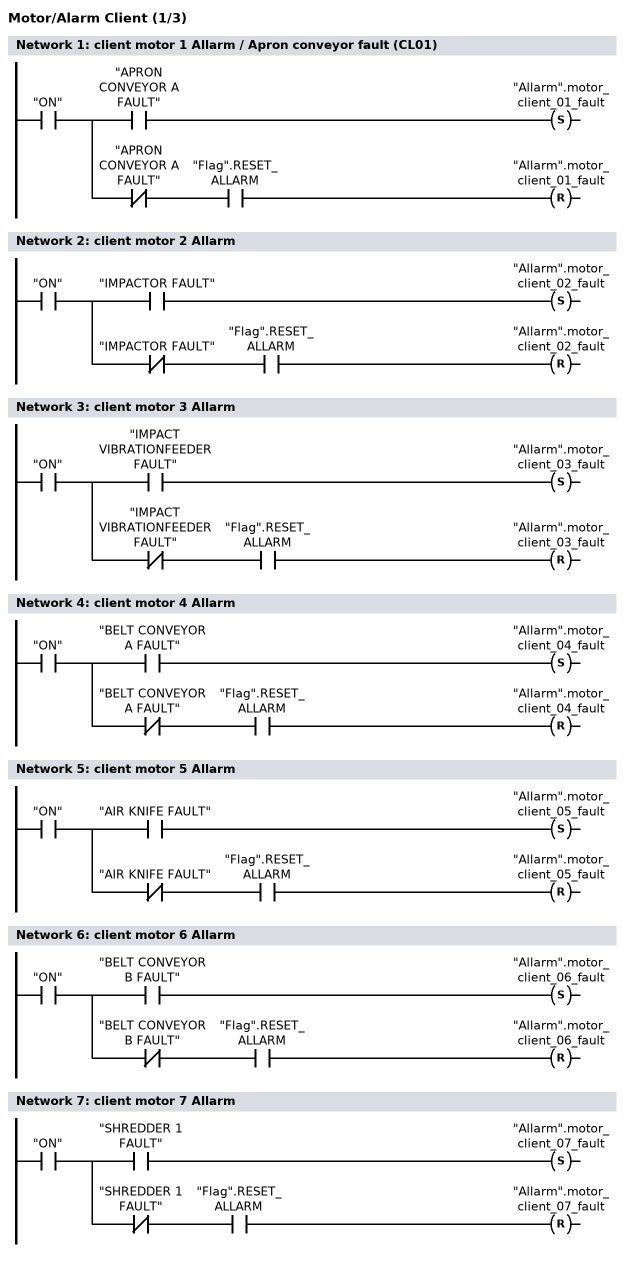
   RUNG wire#powerrail
      Contact( "ON" )
      wire#w1
      Contact( "APRON CONVEYOR A FAULT" )
      S_Coil( "Allarm".motor_client_01_fault )
   END_RUNG
   RUNG wire#w1
      I_Contact( "APRON CONVEYOR A FAULT" )
      Contact( "Flag".RESET_ALLARM )
      R_Coil( "Allarm".motor_client_01_fault )
   END_RUNG
   // the same network as SCL:
   IF "ON" AND "APRON CONVEYOR A FAULT" THEN "Allarm".motor_client_01_fault := TRUE; END_IF;
   IF "ON" AND NOT "APRON CONVEYOR A FAULT" AND "Flag".RESET_ALLARM THEN
       "Allarm".motor_client_01_fault := FALSE;
   END_IF;
END_REGION

REGION Network 2: client motor 2 Allarm
   RUNG wire#powerrail
      Contact( "ON" )
      wire#w1
      Contact( "IMPACTOR FAULT" )
      S_Coil( "Allarm".motor_client_02_fault )
   END_RUNG
   RUNG wire#w1
      I_Contact( "IMPACTOR FAULT" )
      Contact( "Flag".RESET_ALLARM )
      R_Coil( "Allarm".motor_client_02_fault )
   END_RUNG
   // the same network as SCL:
   IF "ON" AND "IMPACTOR FAULT" THEN "Allarm".motor_client_02_fault := TRUE; END_IF;
   IF "ON" AND NOT "IMPACTOR FAULT" AND "Flag".RESET_ALLARM THEN
       "Allarm".motor_client_02_fault := FALSE;
   END_IF;
END_REGION

REGION Network 3: client motor 3 Allarm
   RUNG wire#powerrail
      Contact( "ON" )
      wire#w1
      Contact( "IMPACT VIBRATIONFEEDER FAULT" )
      S_Coil( "Allarm".motor_client_03_fault )
   END_RUNG
   RUNG wire#w1
      I_Contact( "IMPACT VIBRATIONFEEDER FAULT" )
      Contact( "Flag".RESET_ALLARM )
      R_Coil( "Allarm".motor_client_03_fault )
   END_RUNG
   // the same network as SCL:
   IF "ON" AND "IMPACT VIBRATIONFEEDER FAULT" THEN "Allarm".motor_client_03_fault := TRUE; END_IF;
   IF "ON" AND NOT "IMPACT VIBRATIONFEEDER FAULT" AND "Flag".RESET_ALLARM THEN
       "Allarm".motor_client_03_fault := FALSE;
   END_IF;
END_REGION

REGION Network 4: client motor 4 Allarm
   RUNG wire#powerrail
      Contact( "ON" )
      wire#w1
      Contact( "BELT CONVEYOR  A FAULT" )
      S_Coil( "Allarm".motor_client_04_fault )
   END_RUNG
   RUNG wire#w1
      I_Contact( "BELT CONVEYOR  A FAULT" )
      Contact( "Flag".RESET_ALLARM )
      R_Coil( "Allarm".motor_client_04_fault )
   END_RUNG
   // the same network as SCL:
   IF "ON" AND "BELT CONVEYOR  A FAULT" THEN "Allarm".motor_client_04_fault := TRUE; END_IF;
   IF "ON" AND NOT "BELT CONVEYOR  A FAULT" AND "Flag".RESET_ALLARM THEN
       "Allarm".motor_client_04_fault := FALSE;
   END_IF;
END_REGION

REGION Network 5: client motor 5 Allarm
   RUNG wire#powerrail
      Contact( "ON" )
      wire#w1
      Contact( "AIR KNIFE FAULT" )
      S_Coil( "Allarm".motor_client_05_fault )
   END_RUNG
   RUNG wire#w1
      I_Contact( "AIR KNIFE FAULT" )
      Contact( "Flag".RESET_ALLARM )
      R_Coil( "Allarm".motor_client_05_fault )
   END_RUNG
   // the same network as SCL:
   IF "ON" AND "AIR KNIFE FAULT" THEN "Allarm".motor_client_05_fault := TRUE; END_IF;
   IF "ON" AND NOT "AIR KNIFE FAULT" AND "Flag".RESET_ALLARM THEN
       "Allarm".motor_client_05_fault := FALSE;
   END_IF;
END_REGION

REGION Network 6: client motor 6 Allarm
   RUNG wire#powerrail
      Contact( "ON" )
      wire#w1
      Contact( "BELT CONVEYOR B FAULT" )
      S_Coil( "Allarm".motor_client_06_fault )
   END_RUNG
   RUNG wire#w1
      I_Contact( "BELT CONVEYOR B FAULT" )
      Contact( "Flag".RESET_ALLARM )
      R_Coil( "Allarm".motor_client_06_fault )
   END_RUNG
   // the same network as SCL:
   IF "ON" AND "BELT CONVEYOR B FAULT" THEN "Allarm".motor_client_06_fault := TRUE; END_IF;
   IF "ON" AND NOT "BELT CONVEYOR B FAULT" AND "Flag".RESET_ALLARM THEN
       "Allarm".motor_client_06_fault := FALSE;
   END_IF;
END_REGION

REGION Network 7: client motor 7 Allarm
   RUNG wire#powerrail
      Contact( "ON" )
      wire#w1
      Contact( "SHREDDER 1 FAULT" )
      S_Coil( "Allarm".motor_client_07_fault )
   END_RUNG
   RUNG wire#w1
      I_Contact( "SHREDDER 1 FAULT" )
      Contact( "Flag".RESET_ALLARM )
      R_Coil( "Allarm".motor_client_07_fault )
   END_RUNG
   // the same network as SCL:
   IF "ON" AND "SHREDDER 1 FAULT" THEN "Allarm".motor_client_07_fault := TRUE; END_IF;
   IF "ON" AND NOT "SHREDDER 1 FAULT" AND "Flag".RESET_ALLARM THEN
       "Allarm".motor_client_07_fault := FALSE;
   END_IF;
END_REGION

REGION Network 8: client motor 8 Allarm
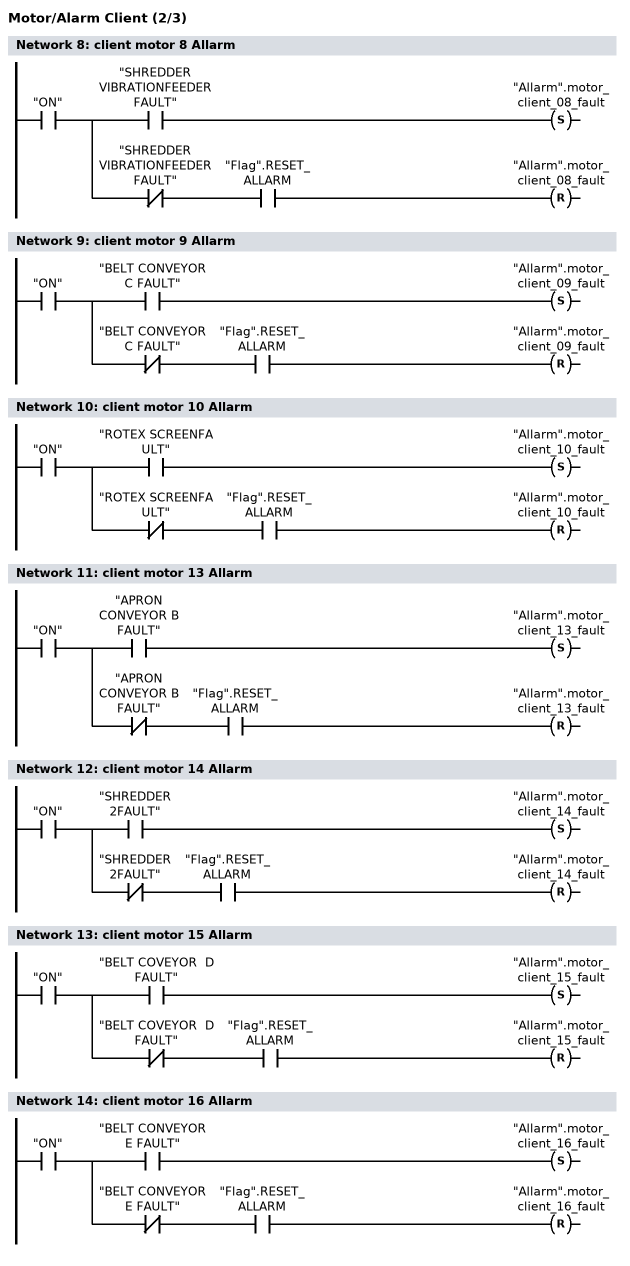
   RUNG wire#powerrail
      Contact( "ON" )
      wire#w1
      Contact( "SHREDDER VIBRATIONFEEDER FAULT" )
      S_Coil( "Allarm".motor_client_08_fault )
   END_RUNG
   RUNG wire#w1
      I_Contact( "SHREDDER VIBRATIONFEEDER FAULT" )
      Contact( "Flag".RESET_ALLARM )
      R_Coil( "Allarm".motor_client_08_fault )
   END_RUNG
   // the same network as SCL:
   IF "ON" AND "SHREDDER VIBRATIONFEEDER FAULT" THEN "Allarm".motor_client_08_fault := TRUE; END_IF;
   IF "ON" AND NOT "SHREDDER VIBRATIONFEEDER FAULT" AND "Flag".RESET_ALLARM THEN
       "Allarm".motor_client_08_fault := FALSE;
   END_IF;
END_REGION

REGION Network 9: client motor 9 Allarm
   RUNG wire#powerrail
      Contact( "ON" )
      wire#w1
      Contact( "BELT CONVEYOR C FAULT" )
      S_Coil( "Allarm".motor_client_09_fault )
   END_RUNG
   RUNG wire#w1
      I_Contact( "BELT CONVEYOR C FAULT" )
      Contact( "Flag".RESET_ALLARM )
      R_Coil( "Allarm".motor_client_09_fault )
   END_RUNG
   // the same network as SCL:
   IF "ON" AND "BELT CONVEYOR C FAULT" THEN "Allarm".motor_client_09_fault := TRUE; END_IF;
   IF "ON" AND NOT "BELT CONVEYOR C FAULT" AND "Flag".RESET_ALLARM THEN
       "Allarm".motor_client_09_fault := FALSE;
   END_IF;
END_REGION

REGION Network 10: client motor 10 Allarm
   RUNG wire#powerrail
      Contact( "ON" )
      wire#w1
      Contact( "ROTEX SCREENFAULT" )
      S_Coil( "Allarm".motor_client_10_fault )
   END_RUNG
   RUNG wire#w1
      I_Contact( "ROTEX SCREENFAULT" )
      Contact( "Flag".RESET_ALLARM )
      R_Coil( "Allarm".motor_client_10_fault )
   END_RUNG
   // the same network as SCL:
   IF "ON" AND "ROTEX SCREENFAULT" THEN "Allarm".motor_client_10_fault := TRUE; END_IF;
   IF "ON" AND NOT "ROTEX SCREENFAULT" AND "Flag".RESET_ALLARM THEN
       "Allarm".motor_client_10_fault := FALSE;
   END_IF;
END_REGION

REGION Network 11: client motor 13 Allarm
   RUNG wire#powerrail
      Contact( "ON" )
      wire#w1
      Contact( "APRON CONVEYOR B FAULT" )
      S_Coil( "Allarm".motor_client_13_fault )
   END_RUNG
   RUNG wire#w1
      I_Contact( "APRON CONVEYOR B FAULT" )
      Contact( "Flag".RESET_ALLARM )
      R_Coil( "Allarm".motor_client_13_fault )
   END_RUNG
   // the same network as SCL:
   IF "ON" AND "APRON CONVEYOR B FAULT" THEN "Allarm".motor_client_13_fault := TRUE; END_IF;
   IF "ON" AND NOT "APRON CONVEYOR B FAULT" AND "Flag".RESET_ALLARM THEN
       "Allarm".motor_client_13_fault := FALSE;
   END_IF;
END_REGION

REGION Network 12: client motor 14 Allarm
   RUNG wire#powerrail
      Contact( "ON" )
      wire#w1
      Contact( "SHREDDER 2FAULT" )
      S_Coil( "Allarm".motor_client_14_fault )
   END_RUNG
   RUNG wire#w1
      I_Contact( "SHREDDER 2FAULT" )
      Contact( "Flag".RESET_ALLARM )
      R_Coil( "Allarm".motor_client_14_fault )
   END_RUNG
   // the same network as SCL:
   IF "ON" AND "SHREDDER 2FAULT" THEN "Allarm".motor_client_14_fault := TRUE; END_IF;
   IF "ON" AND NOT "SHREDDER 2FAULT" AND "Flag".RESET_ALLARM THEN
       "Allarm".motor_client_14_fault := FALSE;
   END_IF;
END_REGION

REGION Network 13: client motor 15 Allarm
   RUNG wire#powerrail
      Contact( "ON" )
      wire#w1
      Contact( "BELT COVEYOR  D FAULT" )
      S_Coil( "Allarm".motor_client_15_fault )
   END_RUNG
   RUNG wire#w1
      I_Contact( "BELT COVEYOR  D FAULT" )
      Contact( "Flag".RESET_ALLARM )
      R_Coil( "Allarm".motor_client_15_fault )
   END_RUNG
   // the same network as SCL:
   IF "ON" AND "BELT COVEYOR  D FAULT" THEN "Allarm".motor_client_15_fault := TRUE; END_IF;
   IF "ON" AND NOT "BELT COVEYOR  D FAULT" AND "Flag".RESET_ALLARM THEN
       "Allarm".motor_client_15_fault := FALSE;
   END_IF;
END_REGION

REGION Network 14: client motor 16 Allarm
   RUNG wire#powerrail
      Contact( "ON" )
      wire#w1
      Contact( "BELT CONVEYOR  E FAULT" )
      S_Coil( "Allarm".motor_client_16_fault )
   END_RUNG
   RUNG wire#w1
      I_Contact( "BELT CONVEYOR  E FAULT" )
      Contact( "Flag".RESET_ALLARM )
      R_Coil( "Allarm".motor_client_16_fault )
   END_RUNG
   // the same network as SCL:
   IF "ON" AND "BELT CONVEYOR  E FAULT" THEN "Allarm".motor_client_16_fault := TRUE; END_IF;
   IF "ON" AND NOT "BELT CONVEYOR  E FAULT" AND "Flag".RESET_ALLARM THEN
       "Allarm".motor_client_16_fault := FALSE;
   END_IF;
END_REGION

REGION Network 15: client motor 17 Allarm
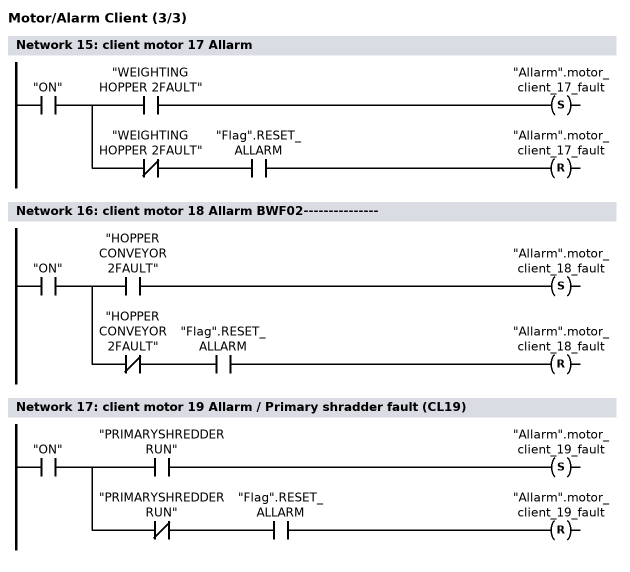
   RUNG wire#powerrail
      Contact( "ON" )
      wire#w1
      Contact( "WEIGHTING HOPPER 2FAULT" )
      S_Coil( "Allarm".motor_client_17_fault )
   END_RUNG
   RUNG wire#w1
      I_Contact( "WEIGHTING HOPPER 2FAULT" )
      Contact( "Flag".RESET_ALLARM )
      R_Coil( "Allarm".motor_client_17_fault )
   END_RUNG
   // the same network as SCL:
   IF "ON" AND "WEIGHTING HOPPER 2FAULT" THEN "Allarm".motor_client_17_fault := TRUE; END_IF;
   IF "ON" AND NOT "WEIGHTING HOPPER 2FAULT" AND "Flag".RESET_ALLARM THEN
       "Allarm".motor_client_17_fault := FALSE;
   END_IF;
END_REGION

REGION Network 16: client motor 18 Allarm BWF02---------------
   RUNG wire#powerrail
      Contact( "ON" )
      wire#w1
      Contact( "HOPPER CONVEYOR 2FAULT" )
      S_Coil( "Allarm".motor_client_18_fault )
   END_RUNG
   RUNG wire#w1
      I_Contact( "HOPPER CONVEYOR 2FAULT" )
      Contact( "Flag".RESET_ALLARM )
      R_Coil( "Allarm".motor_client_18_fault )
   END_RUNG
   // the same network as SCL:
   IF "ON" AND "HOPPER CONVEYOR 2FAULT" THEN "Allarm".motor_client_18_fault := TRUE; END_IF;
   IF "ON" AND NOT "HOPPER CONVEYOR 2FAULT" AND "Flag".RESET_ALLARM THEN
       "Allarm".motor_client_18_fault := FALSE;
   END_IF;
END_REGION

REGION Network 17: client motor 19 Allarm / Primary shradder fault (CL19)
   RUNG wire#powerrail
      Contact( "ON" )
      wire#w1
      Contact( "PRIMARYSHREDDER RUN" )
      S_Coil( "Allarm".motor_client_19_fault )
   END_RUNG
   RUNG wire#w1
      I_Contact( "PRIMARYSHREDDER RUN" )
      Contact( "Flag".RESET_ALLARM )
      R_Coil( "Allarm".motor_client_19_fault )
   END_RUNG
   // the same network as SCL:
   IF "ON" AND "PRIMARYSHREDDER RUN" THEN "Allarm".motor_client_19_fault := TRUE; END_IF;
   IF "ON" AND NOT "PRIMARYSHREDDER RUN" AND "Flag".RESET_ALLARM THEN
       "Allarm".motor_client_19_fault := FALSE;
   END_IF;
END_REGION
END_FUNCTION

FUNCTION "Burner Control" : Void   // FC12, LAD
TITLE = Burner allarms and control
{ S7_Optimized_Access := 'FALSE' }
VERSION : 0.1
   VAR_TEMP
      App00 : Int;
      App01 : Int;
      App02 : Int;
      App03 : Int;
   END_VAR
   VAR_TEMP   // added for the SCL form of the ladder/FBD networks
      _w1 : Bool;
      _w2 : Bool;
      _w3 : Bool;
      _w4 : Bool;
      _w5 : Bool;
      _w6 : Bool;
      _w7 : Bool;
      _w8 : Bool;
      _w9 : Bool;
      _w10 : Bool;
      _w11 : Bool;
   END_VAR
BEGIN

REGION Network 1: Burner box allarm / Burner control box FAULT
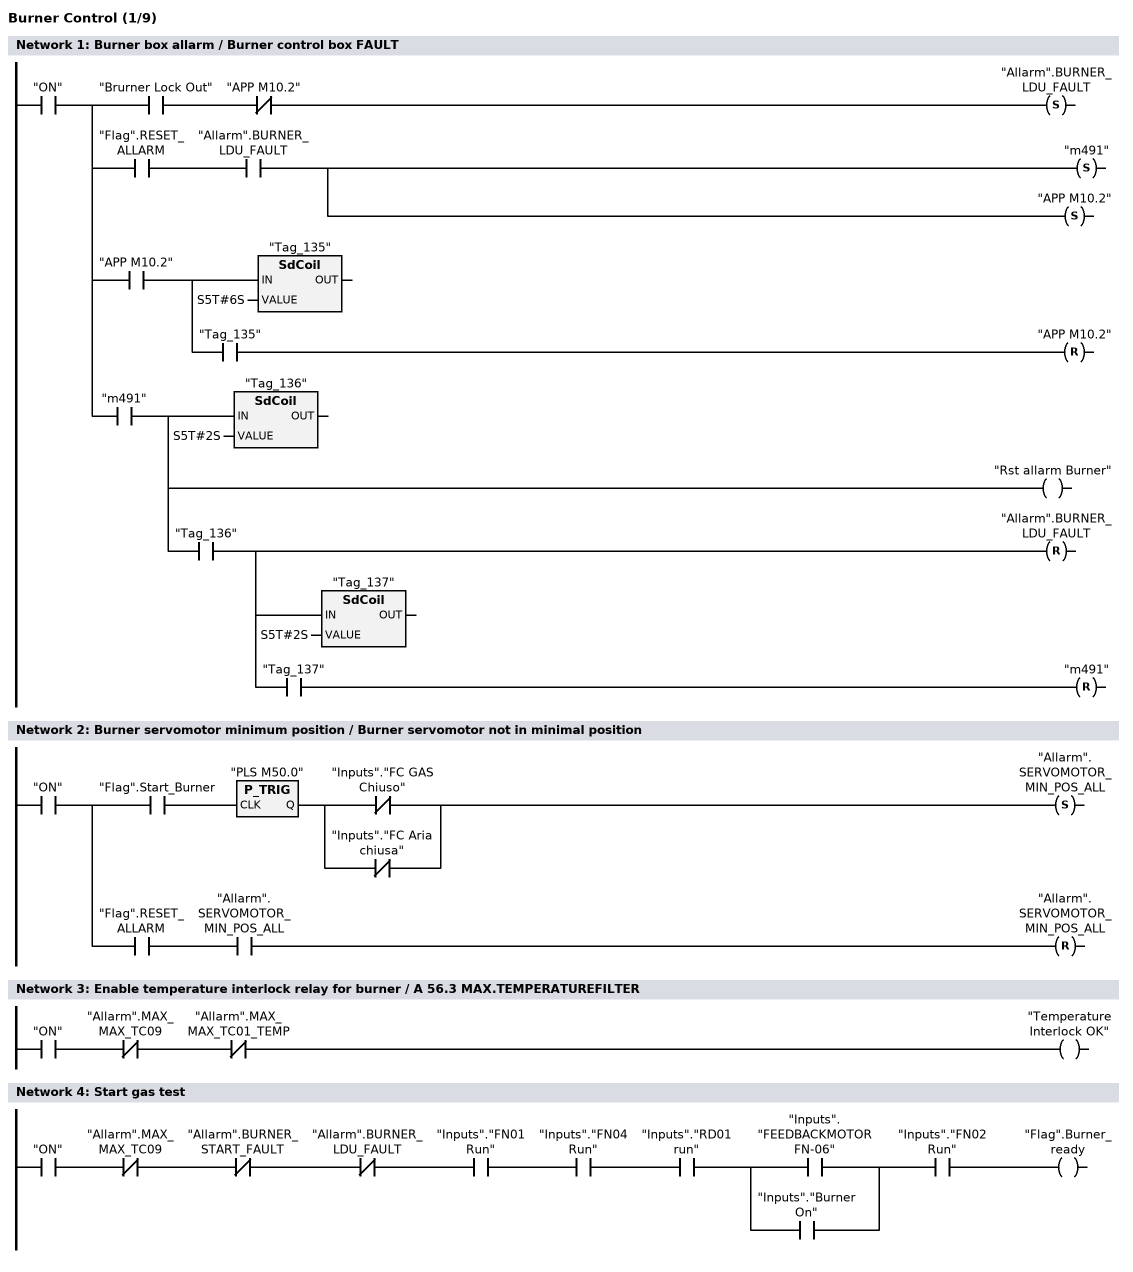
   // no SCL statement known for SdCoil: written as a call
   IF "ON" AND "Brurner Lock Out" AND NOT "APP M10.2" THEN "Allarm".BURNER_LDU_FAULT := TRUE; END_IF;
   IF "ON" AND "Flag".RESET_ALLARM AND "Allarm".BURNER_LDU_FAULT THEN
       "m491" := TRUE;
       "APP M10.2" := TRUE;
   END_IF;
   #_w1 := "ON" AND "APP M10.2";
   #_w2 := "ON";
   SdCoil(in := #_w1, value := S5T#6S, operand := "Tag_135");
   IF #_w1 AND "Tag_135" THEN "APP M10.2" := FALSE; END_IF;
   #_w3 := #_w2 AND "m491";
   SdCoil(in := #_w3, value := S5T#2S, operand := "Tag_136");
   "Rst allarm Burner" := #_w3;
   #_w4 := #_w3 AND "Tag_136";
   IF #_w4 THEN "Allarm".BURNER_LDU_FAULT := FALSE; END_IF;
   SdCoil(in := #_w4, value := S5T#2S, operand := "Tag_137");
   IF #_w4 AND "Tag_137" THEN "m491" := FALSE; END_IF;
END_REGION

REGION Network 2: Burner servomotor minimum position / Burner servomotor not in minimal position
   RUNG wire#powerrail
      Contact( "ON" )
      wire#w1
      Contact( "Flag".Start_Burner )
      P_Trig( "PLS M50.0" )
      wire#w2
      I_Contact( "Inputs"."FC GAS Chiuso" )
      wire#w3
      S_Coil( "Allarm".SERVOMOTOR_MIN_POS_ALL )
   END_RUNG
   RUNG wire#w2
      I_Contact( "Inputs"."FC Aria chiusa" )
   END_RUNG wire#w3
   RUNG wire#w1
      Contact( "Flag".RESET_ALLARM )
      Contact( "Allarm".SERVOMOTOR_MIN_POS_ALL )
      R_Coil( "Allarm".SERVOMOTOR_MIN_POS_ALL )
   END_RUNG
   // the same network as SCL:
   #_w1 := "ON" AND "Flag".Start_Burner;
   #_w2 := #_w1 AND NOT "PLS M50.0";   // rising edge
   "PLS M50.0" := #_w1;
   IF #_w2 AND (NOT "Inputs"."FC GAS Chiuso" OR NOT "Inputs"."FC Aria chiusa") THEN
       "Allarm".SERVOMOTOR_MIN_POS_ALL := TRUE;
   END_IF;
   IF "ON" AND "Flag".RESET_ALLARM AND "Allarm".SERVOMOTOR_MIN_POS_ALL THEN
       "Allarm".SERVOMOTOR_MIN_POS_ALL := FALSE;
   END_IF;
END_REGION

REGION Network 3: Enable temperature interlock relay for burner / A 56.3 MAX.TEMPERATUREFILTER
   RUNG wire#powerrail
      Contact( "ON" )
      I_Contact( "Allarm".MAX_MAX_TC09 )
      I_Contact( "Allarm".MAX_MAX_TC01_TEMP )
      Coil( "Temperature Interlock OK" )
   END_RUNG
   // the same network as SCL:
   "Temperature Interlock OK" := "ON" AND NOT "Allarm".MAX_MAX_TC09 AND NOT "Allarm".MAX_MAX_TC01_TEMP;
END_REGION

REGION Network 4: Start gas test
   RUNG wire#powerrail
      Contact( "ON" )
      I_Contact( "Allarm".MAX_MAX_TC09 )
      I_Contact( "Allarm".BURNER_START_FAULT )
      I_Contact( "Allarm".BURNER_LDU_FAULT )
      Contact( "Inputs"."FN01 Run" )
      Contact( "Inputs"."FN04 Run" )
      Contact( "Inputs"."RD01 run" )
      wire#w1
      Contact( "Inputs"."FEEDBACKMOTOR FN-06" )
      wire#w2
      Contact( "Inputs"."FN02 Run" )
      Coil( "Flag".Burner_ready )
   END_RUNG
   RUNG wire#w1
      Contact( "Inputs"."Burner On" )
   END_RUNG wire#w2
   // the same network as SCL:
   "Flag".Burner_ready := "ON" AND NOT "Allarm".MAX_MAX_TC09 AND NOT "Allarm".BURNER_START_FAULT AND NOT "Allarm".BURNER_LDU_FAULT AND "Inputs"."FN01 Run" AND "Inputs"."FN04 Run" AND "Inputs"."RD01 run" AND ("Inputs"."FEEDBACKMOTOR FN-06" OR "Inputs"."Burner On") AND "Inputs"."FN02 Run";
END_REGION

REGION Network 5: Burner stop
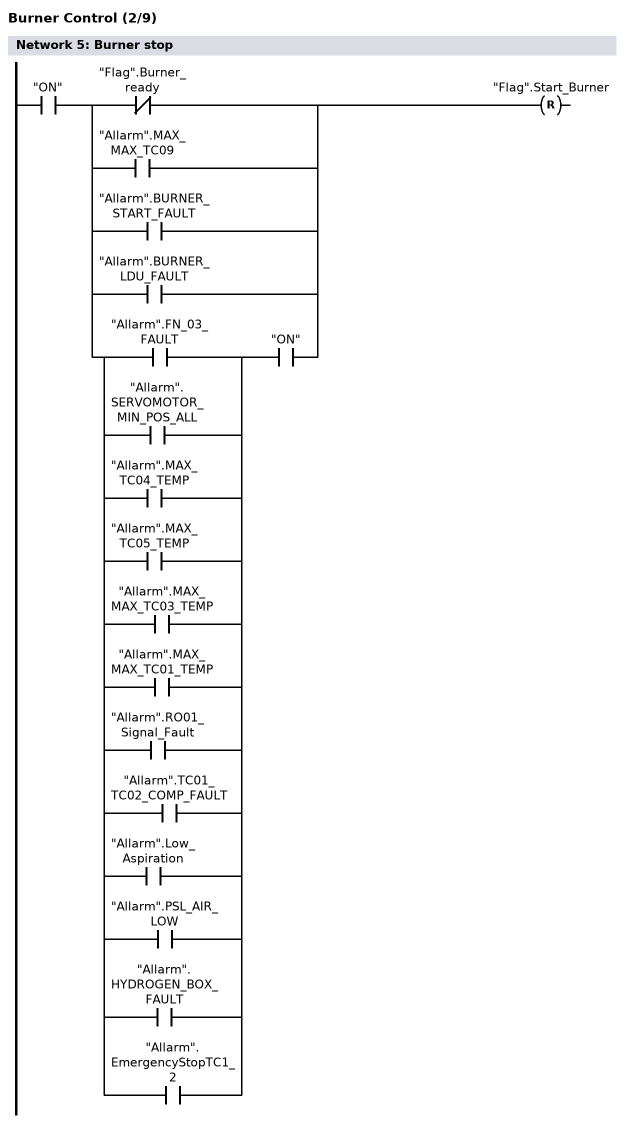
   RUNG wire#powerrail
      Contact( "ON" )
      wire#w1
      I_Contact( "Flag".Burner_ready )
      wire#w2
      R_Coil( "Flag".Start_Burner )
   END_RUNG
   RUNG wire#w1
      Contact( "Allarm".MAX_MAX_TC09 )
   END_RUNG wire#w2
   RUNG wire#w1
      Contact( "Allarm".BURNER_START_FAULT )
   END_RUNG wire#w2
   RUNG wire#w1
      Contact( "Allarm".BURNER_LDU_FAULT )
   END_RUNG wire#w2
   RUNG wire#w1
      Contact( "Allarm".FN_03_FAULT )
      wire#w3
      Contact( "ON" )
   END_RUNG wire#w2
   RUNG wire#w1
      Contact( "Allarm".SERVOMOTOR_MIN_POS_ALL )
   END_RUNG wire#w3
   RUNG wire#w1
      Contact( "Allarm".MAX_TC04_TEMP )
   END_RUNG wire#w3
   RUNG wire#w1
      Contact( "Allarm".MAX_TC05_TEMP )
   END_RUNG wire#w3
   RUNG wire#w1
      Contact( "Allarm".MAX_MAX_TC03_TEMP )
   END_RUNG wire#w3
   RUNG wire#w1
      Contact( "Allarm".MAX_MAX_TC01_TEMP )
   END_RUNG wire#w3
   RUNG wire#w1
      Contact( "Allarm".RO01_Signal_Fault )
   END_RUNG wire#w3
   RUNG wire#w1
      Contact( "Allarm".TC01_TC02_COMP_FAULT )
   END_RUNG wire#w3
   RUNG wire#w1
      Contact( "Allarm".Low_Aspiration )
   END_RUNG wire#w3
   RUNG wire#w1
      Contact( "Allarm".PSL_AIR_LOW )
   END_RUNG wire#w3
   RUNG wire#w1
      Contact( "Allarm".HYDROGEN_BOX_FAULT )
   END_RUNG wire#w3
   RUNG wire#w1
      Contact( "Allarm".EmergencyStopTC1_2 )
   END_RUNG wire#w3
   // the same network as SCL:
   IF "ON" AND (NOT "Flag".Burner_ready OR "Allarm".MAX_MAX_TC09 OR "Allarm".BURNER_START_FAULT OR "Allarm".BURNER_LDU_FAULT OR (("Allarm".FN_03_FAULT OR "Allarm".SERVOMOTOR_MIN_POS_ALL OR "Allarm".MAX_TC04_TEMP OR "Allarm".MAX_TC05_TEMP OR "Allarm".MAX_MAX_TC03_TEMP OR "Allarm".MAX_MAX_TC01_TEMP OR "Allarm".RO01_Signal_Fault OR "Allarm".TC01_TC02_COMP_FAULT OR "Allarm".Low_Aspiration OR "Allarm".PSL_AIR_LOW OR "Allarm".HYDROGEN_BOX_FAULT OR "Allarm".EmergencyStopTC1_2) AND "ON")) THEN
       "Flag".Start_Burner := FALSE;
   END_IF;
END_REGION

REGION Network 6: Conteggio minuti lavoro bruciatore / Counter minutes of burner work
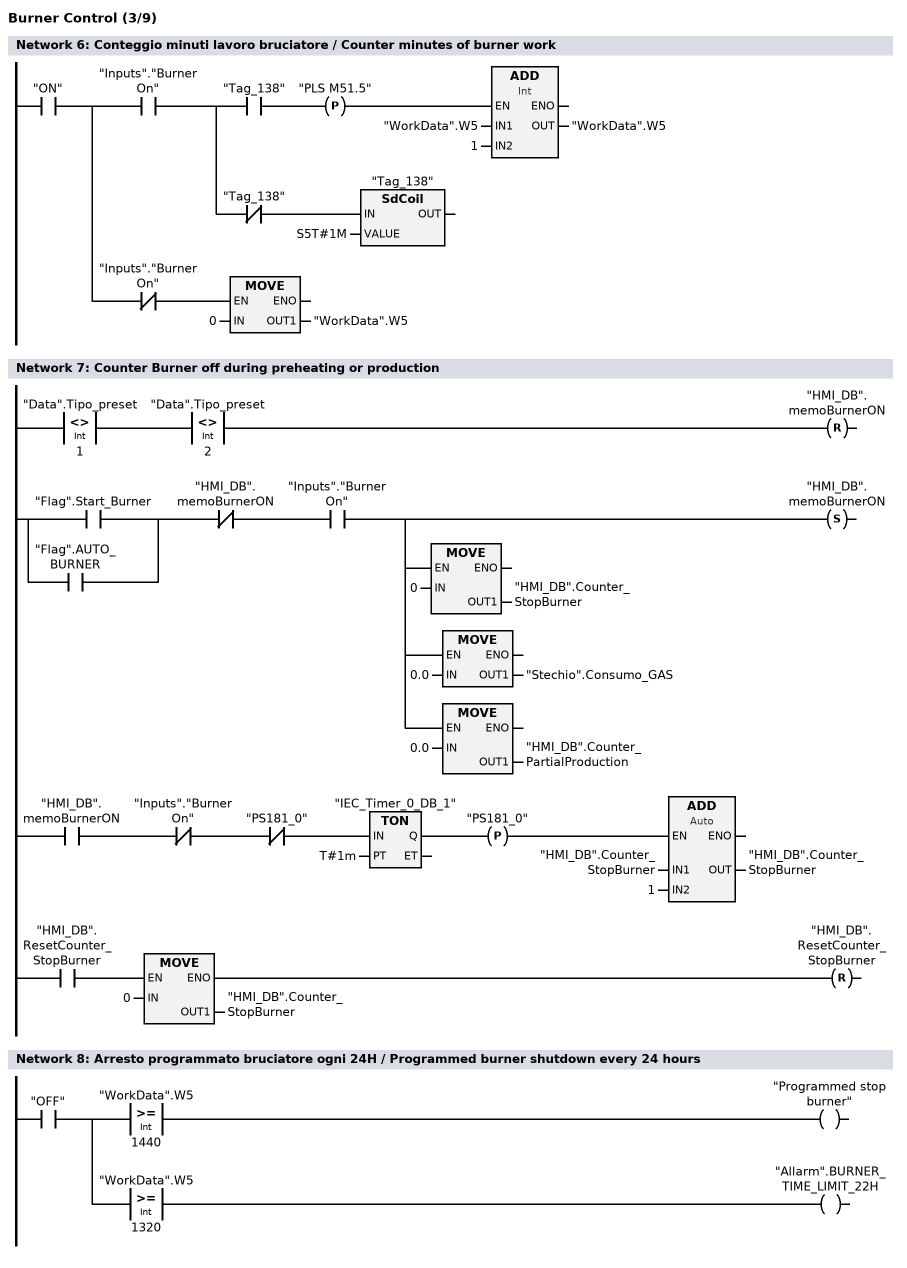
   // no SCL statement known for SdCoil: written as a call
   #_w1 := "ON" AND "Inputs"."Burner On";
   #_w2 := #_w1 AND "Tag_138";
   #_w3 := #_w2 AND NOT "PLS M51.5";   // rising edge
   "PLS M51.5" := #_w2;
   IF #_w3 THEN "WorkData".W5 := "WorkData".W5 + 1; END_IF;
   #_w4 := "ON";
   SdCoil(in := #_w1 AND NOT "Tag_138", value := S5T#1M, operand := "Tag_138");
   IF #_w4 AND NOT "Inputs"."Burner On" THEN "WorkData".W5 := 0; END_IF;
END_REGION

REGION Network 7: Counter Burner off during preheating or production
   IF ("Data".Tipo_preset <> 1) AND ("Data".Tipo_preset <> 2) THEN "HMI_DB".memoBurnerON := FALSE; END_IF;
   #_w1 := ("Flag".Start_Burner OR "Flag".AUTO_BURNER) AND NOT "HMI_DB".memoBurnerON AND "Inputs"."Burner On";
   IF #_w1 THEN
       "HMI_DB".memoBurnerON := TRUE;
       "HMI_DB".Counter_StopBurner := 0;
       "Stechio".Consumo_GAS := 0.0;
       "HMI_DB".Counter_PartialProduction := 0.0;
   END_IF;
   "IEC_Timer_0_DB_1".TON(IN := "HMI_DB".memoBurnerON AND NOT "Inputs"."Burner On" AND NOT "PS181_0",
                          PT := T#1m);
   #_w2 := "IEC_Timer_0_DB_1".Q AND NOT "PS181_0";   // rising edge
   "PS181_0" := "IEC_Timer_0_DB_1".Q;
   IF #_w2 THEN "HMI_DB".Counter_StopBurner := "HMI_DB".Counter_StopBurner + 1; END_IF;
   IF "HMI_DB".ResetCounter_StopBurner THEN
       "HMI_DB".Counter_StopBurner := 0;
       "HMI_DB".ResetCounter_StopBurner := FALSE;
   END_IF;
END_REGION

REGION Network 8: Arresto programmato bruciatore ogni 24H / Programmed burner shutdown every 24 hours
   RUNG wire#powerrail
      Contact( "OFF" )
      wire#w1
      { S7_Templates := "SrcType := Int" } GE_Contact(in1 := "WorkData".W5, in2 := 1440)
      Coil( "Programmed stop burner" )
   END_RUNG
   RUNG wire#w1
      { S7_Templates := "SrcType := Int" } GE_Contact(in1 := "WorkData".W5, in2 := 1320)
      Coil( "Allarm".BURNER_TIME_LIMIT_22H )
   END_RUNG
   // the same network as SCL:
   "Programmed stop burner" := "OFF" AND ("WorkData".W5 >= 1440);
   "Allarm".BURNER_TIME_LIMIT_22H := "OFF" AND ("WorkData".W5 >= 1320);
END_REGION

REGION Network 9: Spegnimento valvola GAS principale se TC01 > 20°C il setpointdb0 / A 56.6 START HIGH FLAMEBURNER
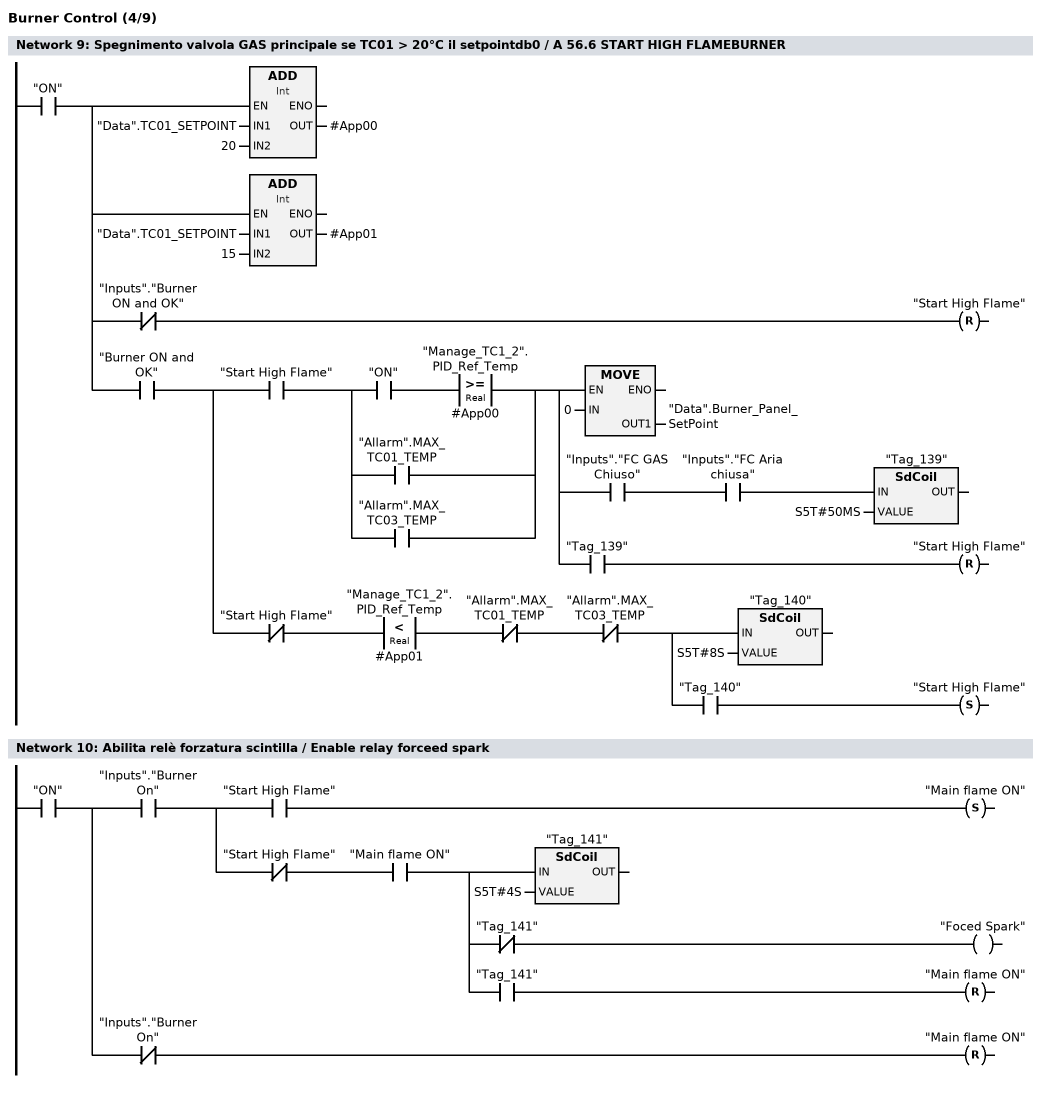
   // no SCL statement known for SdCoil: written as a call
   IF "ON" THEN
       #App00 := "Data".TC01_SETPOINT + 20;
       #App01 := "Data".TC01_SETPOINT + 15;
   END_IF;
   IF "ON" AND NOT "Inputs"."Burner ON and OK" THEN "Start High Flame" := FALSE; END_IF;
   #_w1 := "ON" AND "Burner ON and OK";
   #_w2 := #_w1 AND "Start High Flame" AND (("ON" AND ("Manage_TC1_2".PID_Ref_Temp >= #App00)) OR "Allarm".MAX_TC01_TEMP OR "Allarm".MAX_TC03_TEMP);
   IF #_w2 THEN "Data".Burner_Panel_SetPoint := 0; END_IF;
   SdCoil(in := #_w2 AND "Inputs"."FC GAS Chiuso" AND "Inputs"."FC Aria chiusa",
          value := S5T#50MS,
          operand := "Tag_139");
   IF #_w2 AND "Tag_139" THEN "Start High Flame" := FALSE; END_IF;
   #_w3 := #_w1 AND NOT "Start High Flame" AND ("Manage_TC1_2".PID_Ref_Temp < #App01) AND NOT "Allarm".MAX_TC01_TEMP AND NOT "Allarm".MAX_TC03_TEMP;
   SdCoil(in := #_w3, value := S5T#8S, operand := "Tag_140");
   IF #_w3 AND "Tag_140" THEN "Start High Flame" := TRUE; END_IF;
END_REGION

REGION Network 10: Abilita relè forzatura scintilla / Enable relay forceed spark
   // no SCL statement known for SdCoil: written as a call
   #_w1 := "ON" AND "Inputs"."Burner On";
   IF #_w1 AND "Start High Flame" THEN "Main flame ON" := TRUE; END_IF;
   #_w2 := #_w1 AND NOT "Start High Flame" AND "Main flame ON";
   #_w3 := "ON";
   SdCoil(in := #_w2, value := S5T#4S, operand := "Tag_141");
   "Foced Spark" := #_w2 AND NOT "Tag_141";
   IF #_w2 AND "Tag_141" THEN "Main flame ON" := FALSE; END_IF;
   IF #_w3 AND NOT "Inputs"."Burner On" THEN "Main flame ON" := FALSE; END_IF;
END_REGION

REGION Network 11: Riduce velocità MN01 se TC01 > 30°C il setpoint / reduce speed MN01 se TC01 > 30°C the setpoint
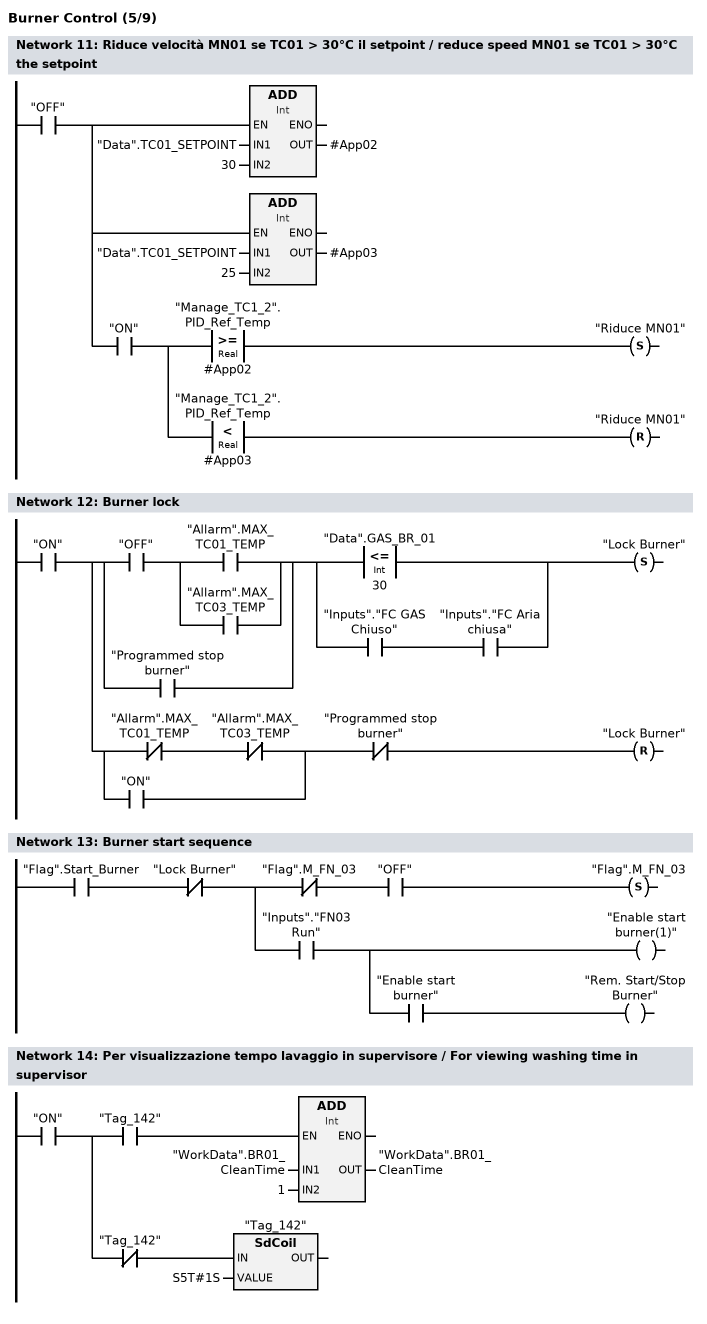
   RUNG wire#powerrail
      Contact( "OFF" )
      wire#w1
      { S7_Templates := "SrcType := Int"; S7_GenerateENO := "TRUE" } Add(in1 := "Data".TC01_SETPOINT, in2 := 30, out => #App02)
   END_RUNG
   RUNG wire#w1
      { S7_Templates := "SrcType := Int"; S7_GenerateENO := "TRUE" } Add(in1 := "Data".TC01_SETPOINT, in2 := 25, out => #App03)
   END_RUNG
   RUNG wire#w1
      Contact( "ON" )
      wire#w2
      { S7_Templates := "SrcType := Real" } GE_Contact(in1 := "Manage_TC1_2".PID_Ref_Temp, in2 := #App02)
      S_Coil( "Riduce MN01" )
   END_RUNG
   RUNG wire#w2
      { S7_Templates := "SrcType := Real" } LT_Contact(in1 := "Manage_TC1_2".PID_Ref_Temp, in2 := #App03)
      R_Coil( "Riduce MN01" )
   END_RUNG
   // the same network as SCL:
   IF "OFF" THEN
       #App02 := "Data".TC01_SETPOINT + 30;
       #App03 := "Data".TC01_SETPOINT + 25;
   END_IF;
   #_w1 := "OFF" AND "ON";
   IF #_w1 AND ("Manage_TC1_2".PID_Ref_Temp >= #App02) THEN "Riduce MN01" := TRUE; END_IF;
   IF #_w1 AND ("Manage_TC1_2".PID_Ref_Temp < #App03) THEN "Riduce MN01" := FALSE; END_IF;
END_REGION

REGION Network 12: Burner lock
   RUNG wire#powerrail
      Contact( "ON" )
      wire#w1
      Contact( "OFF" )
      wire#w2
      Contact( "Allarm".MAX_TC01_TEMP )
      wire#w3
      { S7_Templates := "SrcType := Int" } LE_Contact(in1 := "Data".GAS_BR_01, in2 := 30)
      wire#w4
      S_Coil( "Lock Burner" )
   END_RUNG
   RUNG wire#w2
      Contact( "Allarm".MAX_TC03_TEMP )
   END_RUNG wire#w3
   RUNG wire#w1
      Contact( "Programmed stop burner" )
   END_RUNG wire#w3
   RUNG wire#w3
      Contact( "Inputs"."FC GAS Chiuso" )
      Contact( "Inputs"."FC Aria chiusa" )
   END_RUNG wire#w4
   RUNG wire#w1
      I_Contact( "Allarm".MAX_TC01_TEMP )
      I_Contact( "Allarm".MAX_TC03_TEMP )
      wire#w5
      I_Contact( "Programmed stop burner" )
      R_Coil( "Lock Burner" )
   END_RUNG
   RUNG wire#w1
      Contact( "ON" )
   END_RUNG wire#w5
   // the same network as SCL:
   IF "ON" AND (("OFF" AND ("Allarm".MAX_TC01_TEMP OR "Allarm".MAX_TC03_TEMP)) OR "Programmed stop burner") AND (("Data".GAS_BR_01 <= 30) OR ("Inputs"."FC GAS Chiuso" AND "Inputs"."FC Aria chiusa")) THEN
       "Lock Burner" := TRUE;
   END_IF;
   IF "ON" AND ((NOT "Allarm".MAX_TC01_TEMP AND NOT "Allarm".MAX_TC03_TEMP) OR "ON") AND NOT "Programmed stop burner" THEN
       "Lock Burner" := FALSE;
   END_IF;
END_REGION

REGION Network 13: Burner start sequence
   RUNG wire#powerrail
      Contact( "Flag".Start_Burner )
      I_Contact( "Lock Burner" )
      wire#w1
      I_Contact( "Flag".M_FN_03 )
      Contact( "OFF" )
      S_Coil( "Flag".M_FN_03 )
   END_RUNG
   RUNG wire#w1
      Contact( "Inputs"."FN03 Run" )
      wire#w2
      Coil( "Enable start burner(1)" )
   END_RUNG
   RUNG wire#w2
      Contact( "Enable start burner" )
      Coil( "Rem. Start/Stop Burner" )
   END_RUNG
   // the same network as SCL:
   #_w1 := "Flag".Start_Burner AND NOT "Lock Burner";
   IF #_w1 AND NOT "Flag".M_FN_03 AND "OFF" THEN "Flag".M_FN_03 := TRUE; END_IF;
   "Enable start burner(1)" := #_w1 AND "Inputs"."FN03 Run";
   "Rem. Start/Stop Burner" := "Enable start burner(1)" AND "Enable start burner";
END_REGION

REGION Network 14: Per visualizzazione tempo lavaggio in supervisore / For viewing washing time in supervisor
   // no SCL statement known for SdCoil: written as a call
   IF "ON" AND "Tag_142" THEN "WorkData".BR01_CleanTime := "WorkData".BR01_CleanTime + 1; END_IF;
   SdCoil(in := "ON" AND NOT "Tag_142", value := S5T#1S, operand := "Tag_142");
END_REGION

REGION Network 15: Enable burner cleaning sequence
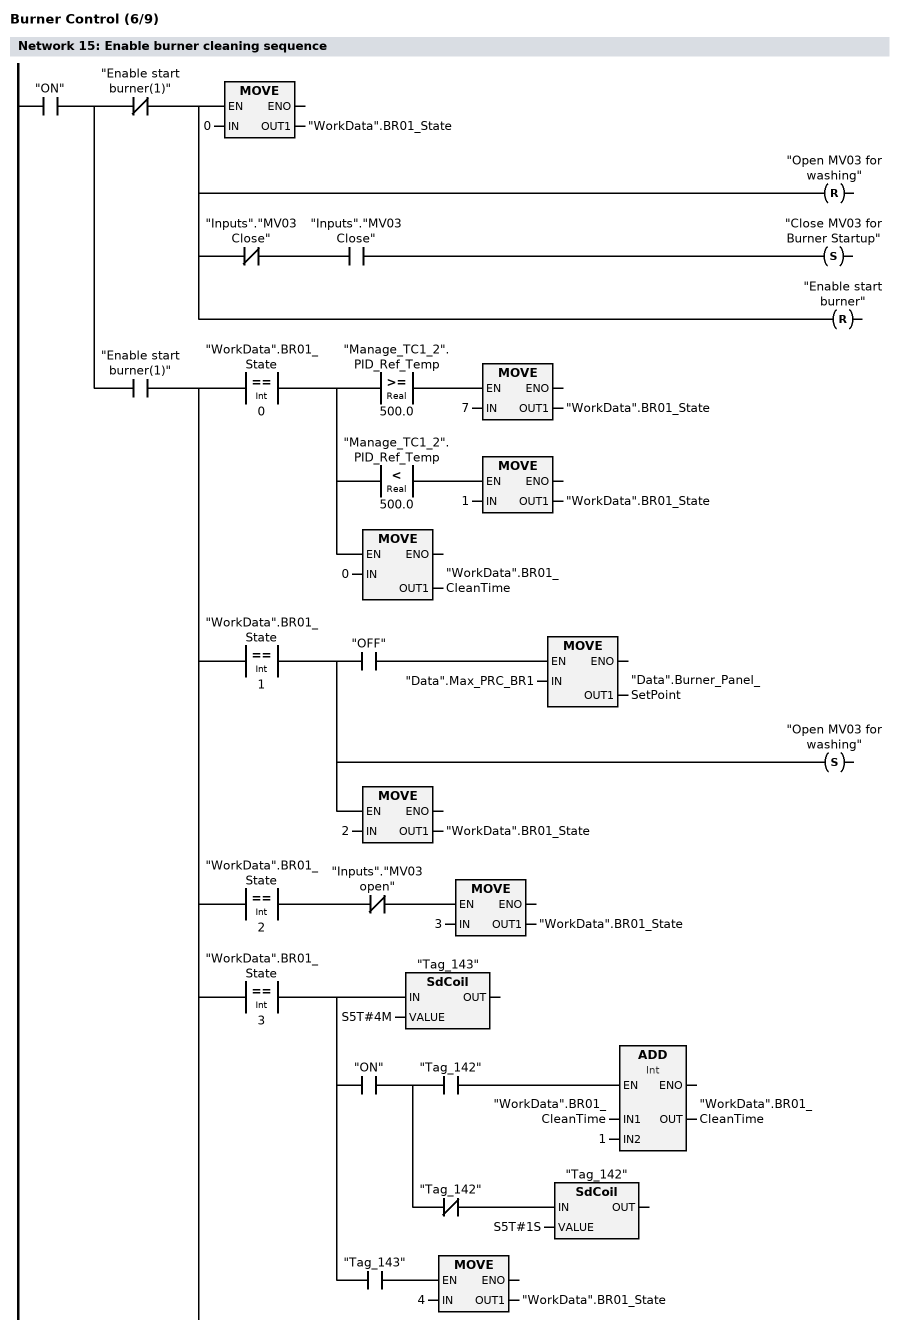
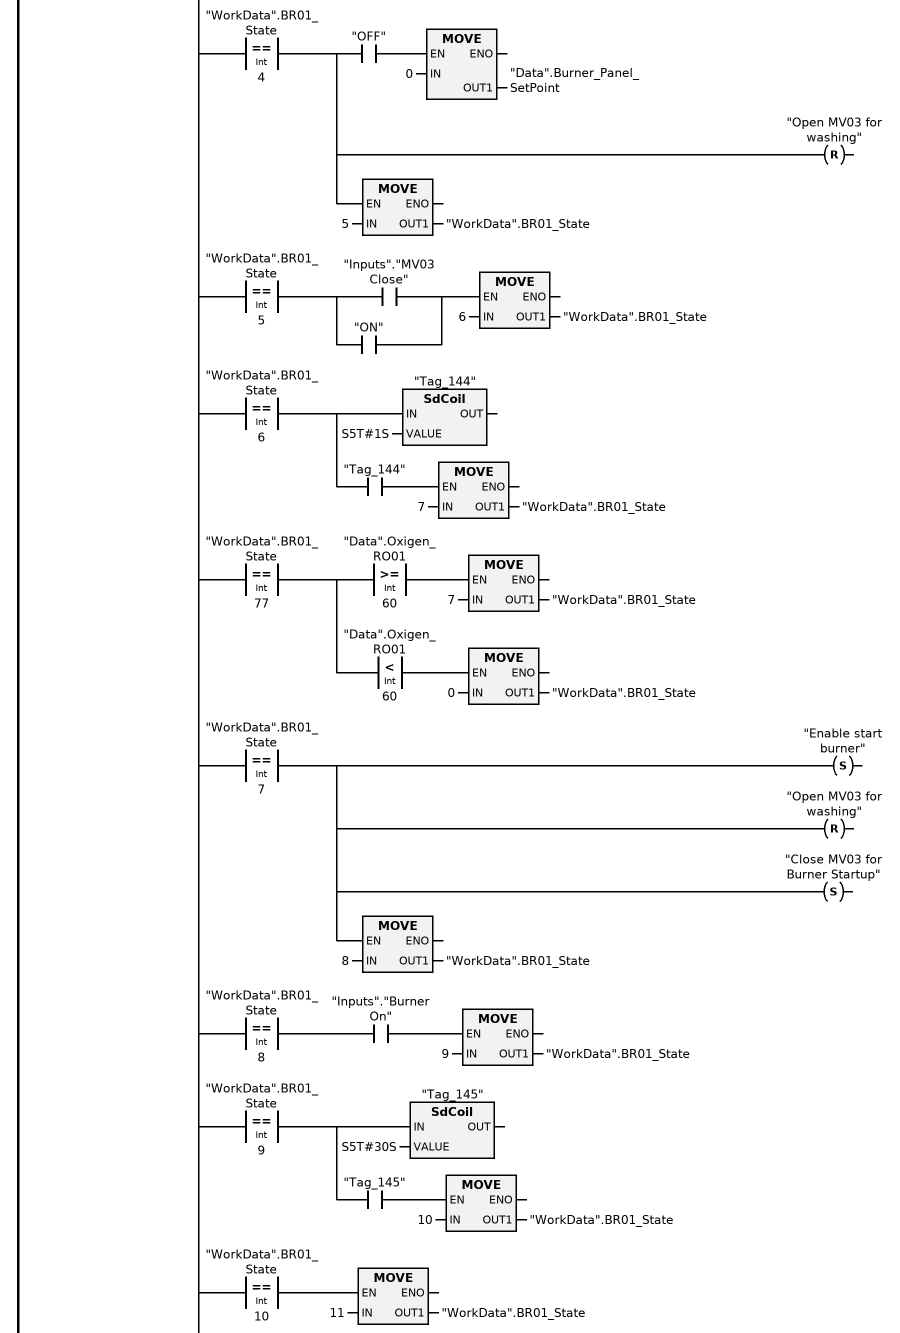
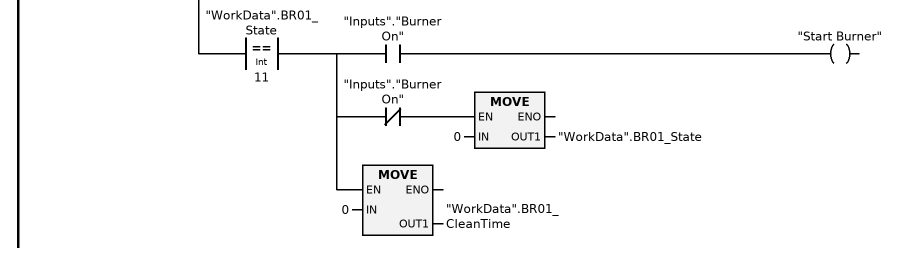
   // no SCL statement known for SdCoil: written as a call
   #_w1 := "ON" AND NOT "Enable start burner(1)";
   IF #_w1 THEN
       "WorkData".BR01_State := 0;
       "Open MV03 for washing" := FALSE;
   END_IF;
   IF #_w1 AND NOT "Inputs"."MV03 Close" AND "Inputs"."MV03 Close" THEN
       "Close MV03 for Burner Startup" := TRUE;
   END_IF;
   IF #_w1 THEN "Enable start burner" := FALSE; END_IF;
   #_w2 := "ON" AND "Enable start burner(1)";
   #_w3 := #_w2 AND ("WorkData".BR01_State = 0);
   IF #_w3 AND ("Manage_TC1_2".PID_Ref_Temp >= 500.0) THEN "WorkData".BR01_State := 7; END_IF;
   IF #_w3 AND ("Manage_TC1_2".PID_Ref_Temp < 500.0) THEN "WorkData".BR01_State := 1; END_IF;
   IF #_w3 THEN "WorkData".BR01_CleanTime := 0; END_IF;
   #_w4 := #_w2 AND ("WorkData".BR01_State = 1);
   IF #_w4 AND "OFF" THEN "Data".Burner_Panel_SetPoint := "Data".Max_PRC_BR1; END_IF;
   IF #_w4 THEN
       "Open MV03 for washing" := TRUE;
       "WorkData".BR01_State := 2;
   END_IF;
   IF #_w2 AND ("WorkData".BR01_State = 2) AND NOT "Inputs"."MV03 open" THEN
       "WorkData".BR01_State := 3;
   END_IF;
   #_w5 := #_w2 AND ("WorkData".BR01_State = 3);
   SdCoil(in := #_w5, value := S5T#4M, operand := "Tag_143");
   #_w6 := #_w5 AND "ON";
   IF #_w6 AND "Tag_142" THEN "WorkData".BR01_CleanTime := "WorkData".BR01_CleanTime + 1; END_IF;
   SdCoil(in := #_w6 AND NOT "Tag_142", value := S5T#1S, operand := "Tag_142");
   IF #_w5 AND "Tag_143" THEN "WorkData".BR01_State := 4; END_IF;
   #_w7 := #_w2 AND ("WorkData".BR01_State = 4);
   IF #_w7 AND "OFF" THEN "Data".Burner_Panel_SetPoint := 0; END_IF;
   IF #_w7 THEN
       "Open MV03 for washing" := FALSE;
       "WorkData".BR01_State := 5;
   END_IF;
   IF #_w2 AND ("WorkData".BR01_State = 5) AND ("Inputs"."MV03 Close" OR "ON") THEN
       "WorkData".BR01_State := 6;
   END_IF;
   #_w8 := #_w2 AND ("WorkData".BR01_State = 6);
   SdCoil(in := #_w8, value := S5T#1S, operand := "Tag_144");
   IF #_w8 AND "Tag_144" THEN "WorkData".BR01_State := 7; END_IF;
   #_w9 := #_w2 AND ("WorkData".BR01_State = 77);
   IF #_w9 AND ("Data".Oxigen_RO01 >= 60) THEN "WorkData".BR01_State := 7; END_IF;
   IF #_w9 AND ("Data".Oxigen_RO01 < 60) THEN "WorkData".BR01_State := 0; END_IF;
   IF #_w2 AND ("WorkData".BR01_State = 7) THEN
       "Enable start burner" := TRUE;
       "Open MV03 for washing" := FALSE;
       "Close MV03 for Burner Startup" := TRUE;
       "WorkData".BR01_State := 8;
   END_IF;
   IF #_w2 AND ("WorkData".BR01_State = 8) AND "Inputs"."Burner On" THEN "WorkData".BR01_State := 9; END_IF;
   #_w10 := #_w2 AND ("WorkData".BR01_State = 9);
   SdCoil(in := #_w10, value := S5T#30S, operand := "Tag_145");
   IF #_w10 AND "Tag_145" THEN "WorkData".BR01_State := 10; END_IF;
   IF #_w2 AND ("WorkData".BR01_State = 10) THEN "WorkData".BR01_State := 11; END_IF;
   #_w11 := #_w2 AND ("WorkData".BR01_State = 11);
   "Start Burner" := #_w11 AND "Inputs"."Burner On";
   IF #_w11 AND NOT "Inputs"."Burner On" THEN "WorkData".BR01_State := 0; END_IF;
   IF #_w11 THEN "WorkData".BR01_CleanTime := 0; END_IF;
END_REGION

REGION Network 16: Burner start fault reset
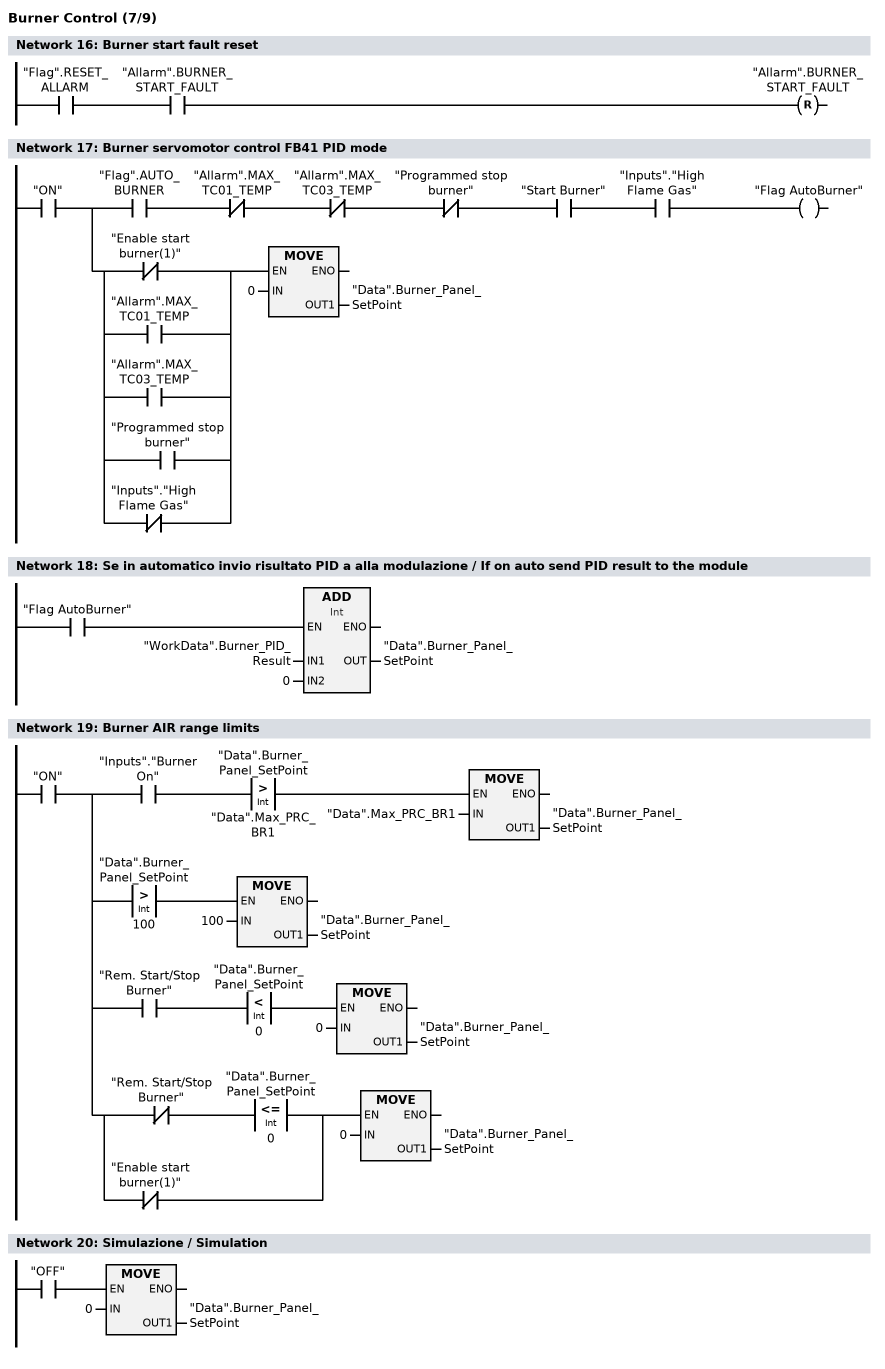
   RUNG wire#powerrail
      Contact( "Flag".RESET_ALLARM )
      Contact( "Allarm".BURNER_START_FAULT )
      R_Coil( "Allarm".BURNER_START_FAULT )
   END_RUNG
   // the same network as SCL:
   IF "Flag".RESET_ALLARM AND "Allarm".BURNER_START_FAULT THEN "Allarm".BURNER_START_FAULT := FALSE; END_IF;
END_REGION

REGION Network 17: Burner servomotor control FB41 PID mode
   RUNG wire#powerrail
      Contact( "ON" )
      wire#w1
      Contact( "Flag".AUTO_BURNER )
      I_Contact( "Allarm".MAX_TC01_TEMP )
      I_Contact( "Allarm".MAX_TC03_TEMP )
      I_Contact( "Programmed stop burner" )
      Contact( "Start Burner" )
      Contact( "Inputs"."High Flame Gas" )
      Coil( "Flag AutoBurner" )
   END_RUNG
   RUNG wire#w1
      I_Contact( "Enable start burner(1)" )
      wire#w2
      { S7_GenerateENO := "TRUE" } Move(in := 0, out1 => "Data".Burner_Panel_SetPoint)
   END_RUNG
   RUNG wire#w1
      Contact( "Allarm".MAX_TC01_TEMP )
   END_RUNG wire#w2
   RUNG wire#w1
      Contact( "Allarm".MAX_TC03_TEMP )
   END_RUNG wire#w2
   RUNG wire#w1
      Contact( "Programmed stop burner" )
   END_RUNG wire#w2
   RUNG wire#w1
      I_Contact( "Inputs"."High Flame Gas" )
   END_RUNG wire#w2
   // the same network as SCL:
   "Flag AutoBurner" := "ON" AND "Flag".AUTO_BURNER AND NOT "Allarm".MAX_TC01_TEMP AND NOT "Allarm".MAX_TC03_TEMP AND NOT "Programmed stop burner" AND "Start Burner" AND "Inputs"."High Flame Gas";
   IF "ON" AND (NOT "Enable start burner(1)" OR "Allarm".MAX_TC01_TEMP OR "Allarm".MAX_TC03_TEMP OR "Programmed stop burner" OR NOT "Inputs"."High Flame Gas") THEN
       "Data".Burner_Panel_SetPoint := 0;
   END_IF;
END_REGION

REGION Network 18: Se in automatico invio risultato PID a alla modulazione / If on auto send PID result to the module
   RUNG wire#powerrail
      Contact( "Flag AutoBurner" )
      { S7_Templates := "SrcType := Int"; S7_GenerateENO := "TRUE" } Add(in1 := "WorkData".Burner_PID_Result, in2 := 0, out => "Data".Burner_Panel_SetPoint)
   END_RUNG
   // the same network as SCL:
   IF "Flag AutoBurner" THEN "Data".Burner_Panel_SetPoint := "WorkData".Burner_PID_Result + 0; END_IF;
END_REGION

REGION Network 19: Burner AIR range limits
   RUNG wire#powerrail
      Contact( "ON" )
      wire#w1
      Contact( "Inputs"."Burner On" )
      { S7_Templates := "SrcType := Int" } GT_Contact(in1 := "Data".Burner_Panel_SetPoint, in2 := "Data".Max_PRC_BR1)
      { S7_GenerateENO := "TRUE" } Move(in := "Data".Max_PRC_BR1, out1 => "Data".Burner_Panel_SetPoint)
   END_RUNG
   RUNG wire#w1
      { S7_Templates := "SrcType := Int" } GT_Contact(in1 := "Data".Burner_Panel_SetPoint, in2 := 100)
      { S7_GenerateENO := "TRUE" } Move(in := 100, out1 => "Data".Burner_Panel_SetPoint)
   END_RUNG
   RUNG wire#w1
      Contact( "Rem. Start/Stop Burner" )
      { S7_Templates := "SrcType := Int" } LT_Contact(in1 := "Data".Burner_Panel_SetPoint, in2 := 0)
      { S7_GenerateENO := "TRUE" } Move(in := 0, out1 => "Data".Burner_Panel_SetPoint)
   END_RUNG
   RUNG wire#w1
      I_Contact( "Rem. Start/Stop Burner" )
      { S7_Templates := "SrcType := Int" } LE_Contact(in1 := "Data".Burner_Panel_SetPoint, in2 := 0)
      wire#w2
      { S7_GenerateENO := "TRUE" } Move(in := 0, out1 => "Data".Burner_Panel_SetPoint)
   END_RUNG
   RUNG wire#w1
      I_Contact( "Enable start burner(1)" )
   END_RUNG wire#w2
   // the same network as SCL:
   IF "ON" AND "Inputs"."Burner On" AND ("Data".Burner_Panel_SetPoint > "Data".Max_PRC_BR1) THEN
       "Data".Burner_Panel_SetPoint := "Data".Max_PRC_BR1;
   END_IF;
   IF "ON" AND ("Data".Burner_Panel_SetPoint > 100) THEN "Data".Burner_Panel_SetPoint := 100; END_IF;
   IF "ON" AND "Rem. Start/Stop Burner" AND ("Data".Burner_Panel_SetPoint < 0) THEN
       "Data".Burner_Panel_SetPoint := 0;
   END_IF;
   IF "ON" AND ((NOT "Rem. Start/Stop Burner" AND ("Data".Burner_Panel_SetPoint <= 0)) OR NOT "Enable start burner(1)") THEN
       "Data".Burner_Panel_SetPoint := 0;
   END_IF;
END_REGION

REGION Network 20: Simulazione / Simulation
   RUNG wire#powerrail
      Contact( "OFF" )
      { S7_GenerateENO := "TRUE" } Move(in := 0, out1 => "Data".Burner_Panel_SetPoint)
   END_RUNG
   // the same network as SCL:
   IF "OFF" THEN "Data".Burner_Panel_SetPoint := 0; END_IF;
END_REGION

REGION Network 21: Genera allarme se persistono limiti di correzione stechiometrica / Stoichiometry out of range
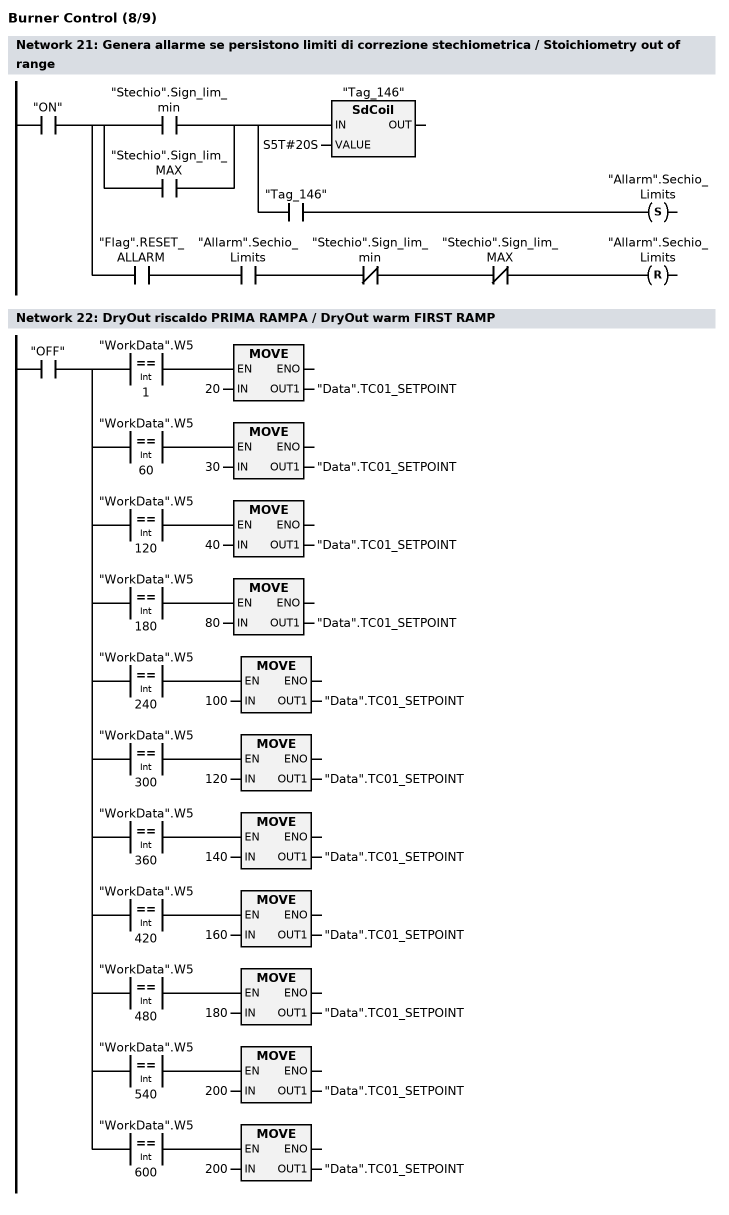
   // no SCL statement known for SdCoil: written as a call
   #_w1 := "ON" AND ("Stechio".Sign_lim_min OR "Stechio".Sign_lim_MAX);
   #_w2 := "ON";
   SdCoil(in := #_w1, value := S5T#20S, operand := "Tag_146");
   IF #_w1 AND "Tag_146" THEN "Allarm".Sechio_Limits := TRUE; END_IF;
   IF #_w2 AND "Flag".RESET_ALLARM AND "Allarm".Sechio_Limits AND NOT "Stechio".Sign_lim_min AND NOT "Stechio".Sign_lim_MAX THEN
       "Allarm".Sechio_Limits := FALSE;
   END_IF;
END_REGION

REGION Network 22: DryOut riscaldo PRIMA RAMPA / DryOut warm FIRST RAMP
   RUNG wire#powerrail
      Contact( "OFF" )
      wire#w1
      { S7_Templates := "SrcType := Int" } EQ_Contact(in1 := "WorkData".W5, in2 := 1)
      { S7_GenerateENO := "TRUE" } Move(in := 20, out1 => "Data".TC01_SETPOINT)
   END_RUNG
   RUNG wire#w1
      { S7_Templates := "SrcType := Int" } EQ_Contact(in1 := "WorkData".W5, in2 := 60)
      { S7_GenerateENO := "TRUE" } Move(in := 30, out1 => "Data".TC01_SETPOINT)
   END_RUNG
   RUNG wire#w1
      { S7_Templates := "SrcType := Int" } EQ_Contact(in1 := "WorkData".W5, in2 := 120)
      { S7_GenerateENO := "TRUE" } Move(in := 40, out1 => "Data".TC01_SETPOINT)
   END_RUNG
   RUNG wire#w1
      { S7_Templates := "SrcType := Int" } EQ_Contact(in1 := "WorkData".W5, in2 := 180)
      { S7_GenerateENO := "TRUE" } Move(in := 80, out1 => "Data".TC01_SETPOINT)
   END_RUNG
   RUNG wire#w1
      { S7_Templates := "SrcType := Int" } EQ_Contact(in1 := "WorkData".W5, in2 := 240)
      { S7_GenerateENO := "TRUE" } Move(in := 100, out1 => "Data".TC01_SETPOINT)
   END_RUNG
   RUNG wire#w1
      { S7_Templates := "SrcType := Int" } EQ_Contact(in1 := "WorkData".W5, in2 := 300)
      { S7_GenerateENO := "TRUE" } Move(in := 120, out1 => "Data".TC01_SETPOINT)
   END_RUNG
   RUNG wire#w1
      { S7_Templates := "SrcType := Int" } EQ_Contact(in1 := "WorkData".W5, in2 := 360)
      { S7_GenerateENO := "TRUE" } Move(in := 140, out1 => "Data".TC01_SETPOINT)
   END_RUNG
   RUNG wire#w1
      { S7_Templates := "SrcType := Int" } EQ_Contact(in1 := "WorkData".W5, in2 := 420)
      { S7_GenerateENO := "TRUE" } Move(in := 160, out1 => "Data".TC01_SETPOINT)
   END_RUNG
   RUNG wire#w1
      { S7_Templates := "SrcType := Int" } EQ_Contact(in1 := "WorkData".W5, in2 := 480)
      { S7_GenerateENO := "TRUE" } Move(in := 180, out1 => "Data".TC01_SETPOINT)
   END_RUNG
   RUNG wire#w1
      { S7_Templates := "SrcType := Int" } EQ_Contact(in1 := "WorkData".W5, in2 := 540)
      { S7_GenerateENO := "TRUE" } Move(in := 200, out1 => "Data".TC01_SETPOINT)
   END_RUNG
   RUNG wire#w1
      { S7_Templates := "SrcType := Int" } EQ_Contact(in1 := "WorkData".W5, in2 := 600)
      { S7_GenerateENO := "TRUE" } Move(in := 200, out1 => "Data".TC01_SETPOINT)
   END_RUNG
   // the same network as SCL:
   IF "OFF" AND ("WorkData".W5 = 1) THEN "Data".TC01_SETPOINT := 20; END_IF;
   IF "OFF" AND ("WorkData".W5 = 60) THEN "Data".TC01_SETPOINT := 30; END_IF;
   IF "OFF" AND ("WorkData".W5 = 120) THEN "Data".TC01_SETPOINT := 40; END_IF;
   IF "OFF" AND ("WorkData".W5 = 180) THEN "Data".TC01_SETPOINT := 80; END_IF;
   IF "OFF" AND ("WorkData".W5 = 240) THEN "Data".TC01_SETPOINT := 100; END_IF;
   IF "OFF" AND ("WorkData".W5 = 300) THEN "Data".TC01_SETPOINT := 120; END_IF;
   IF "OFF" AND ("WorkData".W5 = 360) THEN "Data".TC01_SETPOINT := 140; END_IF;
   IF "OFF" AND ("WorkData".W5 = 420) THEN "Data".TC01_SETPOINT := 160; END_IF;
   IF "OFF" AND ("WorkData".W5 = 480) THEN "Data".TC01_SETPOINT := 180; END_IF;
   IF "OFF" AND ("WorkData".W5 = 540) THEN "Data".TC01_SETPOINT := 200; END_IF;
   IF "OFF" AND ("WorkData".W5 = 600) THEN "Data".TC01_SETPOINT := 200; END_IF;
END_REGION

REGION Network 23: DryOut riscaldo SECONDA RAMPA / DryOut warm SECOND RAMP
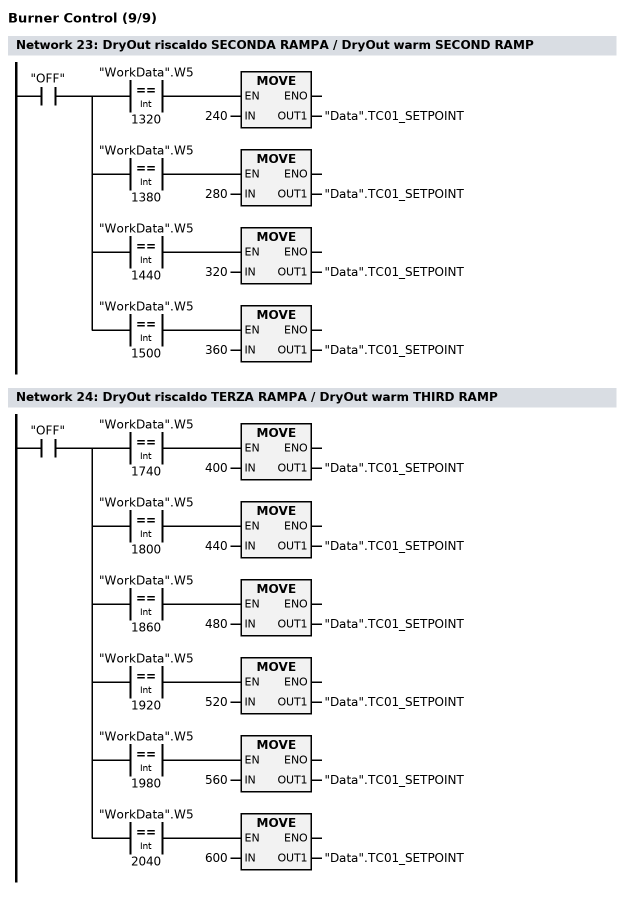
   RUNG wire#powerrail
      Contact( "OFF" )
      wire#w1
      { S7_Templates := "SrcType := Int" } EQ_Contact(in1 := "WorkData".W5, in2 := 1320)
      { S7_GenerateENO := "TRUE" } Move(in := 240, out1 => "Data".TC01_SETPOINT)
   END_RUNG
   RUNG wire#w1
      { S7_Templates := "SrcType := Int" } EQ_Contact(in1 := "WorkData".W5, in2 := 1380)
      { S7_GenerateENO := "TRUE" } Move(in := 280, out1 => "Data".TC01_SETPOINT)
   END_RUNG
   RUNG wire#w1
      { S7_Templates := "SrcType := Int" } EQ_Contact(in1 := "WorkData".W5, in2 := 1440)
      { S7_GenerateENO := "TRUE" } Move(in := 320, out1 => "Data".TC01_SETPOINT)
   END_RUNG
   RUNG wire#w1
      { S7_Templates := "SrcType := Int" } EQ_Contact(in1 := "WorkData".W5, in2 := 1500)
      { S7_GenerateENO := "TRUE" } Move(in := 360, out1 => "Data".TC01_SETPOINT)
   END_RUNG
   // the same network as SCL:
   IF "OFF" AND ("WorkData".W5 = 1320) THEN "Data".TC01_SETPOINT := 240; END_IF;
   IF "OFF" AND ("WorkData".W5 = 1380) THEN "Data".TC01_SETPOINT := 280; END_IF;
   IF "OFF" AND ("WorkData".W5 = 1440) THEN "Data".TC01_SETPOINT := 320; END_IF;
   IF "OFF" AND ("WorkData".W5 = 1500) THEN "Data".TC01_SETPOINT := 360; END_IF;
END_REGION

REGION Network 24: DryOut riscaldo TERZA RAMPA / DryOut warm THIRD RAMP
   RUNG wire#powerrail
      Contact( "OFF" )
      wire#w1
      { S7_Templates := "SrcType := Int" } EQ_Contact(in1 := "WorkData".W5, in2 := 1740)
      { S7_GenerateENO := "TRUE" } Move(in := 400, out1 => "Data".TC01_SETPOINT)
   END_RUNG
   RUNG wire#w1
      { S7_Templates := "SrcType := Int" } EQ_Contact(in1 := "WorkData".W5, in2 := 1800)
      { S7_GenerateENO := "TRUE" } Move(in := 440, out1 => "Data".TC01_SETPOINT)
   END_RUNG
   RUNG wire#w1
      { S7_Templates := "SrcType := Int" } EQ_Contact(in1 := "WorkData".W5, in2 := 1860)
      { S7_GenerateENO := "TRUE" } Move(in := 480, out1 => "Data".TC01_SETPOINT)
   END_RUNG
   RUNG wire#w1
      { S7_Templates := "SrcType := Int" } EQ_Contact(in1 := "WorkData".W5, in2 := 1920)
      { S7_GenerateENO := "TRUE" } Move(in := 520, out1 => "Data".TC01_SETPOINT)
   END_RUNG
   RUNG wire#w1
      { S7_Templates := "SrcType := Int" } EQ_Contact(in1 := "WorkData".W5, in2 := 1980)
      { S7_GenerateENO := "TRUE" } Move(in := 560, out1 => "Data".TC01_SETPOINT)
   END_RUNG
   RUNG wire#w1
      { S7_Templates := "SrcType := Int" } EQ_Contact(in1 := "WorkData".W5, in2 := 2040)
      { S7_GenerateENO := "TRUE" } Move(in := 600, out1 => "Data".TC01_SETPOINT)
   END_RUNG
   // the same network as SCL:
   IF "OFF" AND ("WorkData".W5 = 1740) THEN "Data".TC01_SETPOINT := 400; END_IF;
   IF "OFF" AND ("WorkData".W5 = 1800) THEN "Data".TC01_SETPOINT := 440; END_IF;
   IF "OFF" AND ("WorkData".W5 = 1860) THEN "Data".TC01_SETPOINT := 480; END_IF;
   IF "OFF" AND ("WorkData".W5 = 1920) THEN "Data".TC01_SETPOINT := 520; END_IF;
   IF "OFF" AND ("WorkData".W5 = 1980) THEN "Data".TC01_SETPOINT := 560; END_IF;
   IF "OFF" AND ("WorkData".W5 = 2040) THEN "Data".TC01_SETPOINT := 600; END_IF;
END_REGION
END_FUNCTION

FUNCTION "Control_stechio" : Void   // FC13, LAD
TITLE = Questa FC è eseguita ogni 100ms / This FC is runned every 100ms
{ S7_Optimized_Access := 'FALSE' }
VERSION : 0.1
   VAR_TEMP
      AIR_FLOW : Real;
      GAS_FLOW : Real;
      Correzione_Stechio : Real;
      Correzione_Stechio_INT : Int;
      Portata_Presunta_GAS : Int;
      Portata_Aria_richiesta : Real;
      Correz : Real;
      Correzione_Calcolata_INT : Int;
      Stechio_attuale : Real;
      SetPoint_Stechio : Real;
      Portata_al_secondo : Real;
      AppReal01 : Real;
      PID_TI_S : Time;
      PID_TD_S : Time;
   END_VAR
BEGIN

REGION Network 1: Calcola la portata GAS in base alla rampa teorica / Calculate the GAS flow rate based on the theoretical ramp
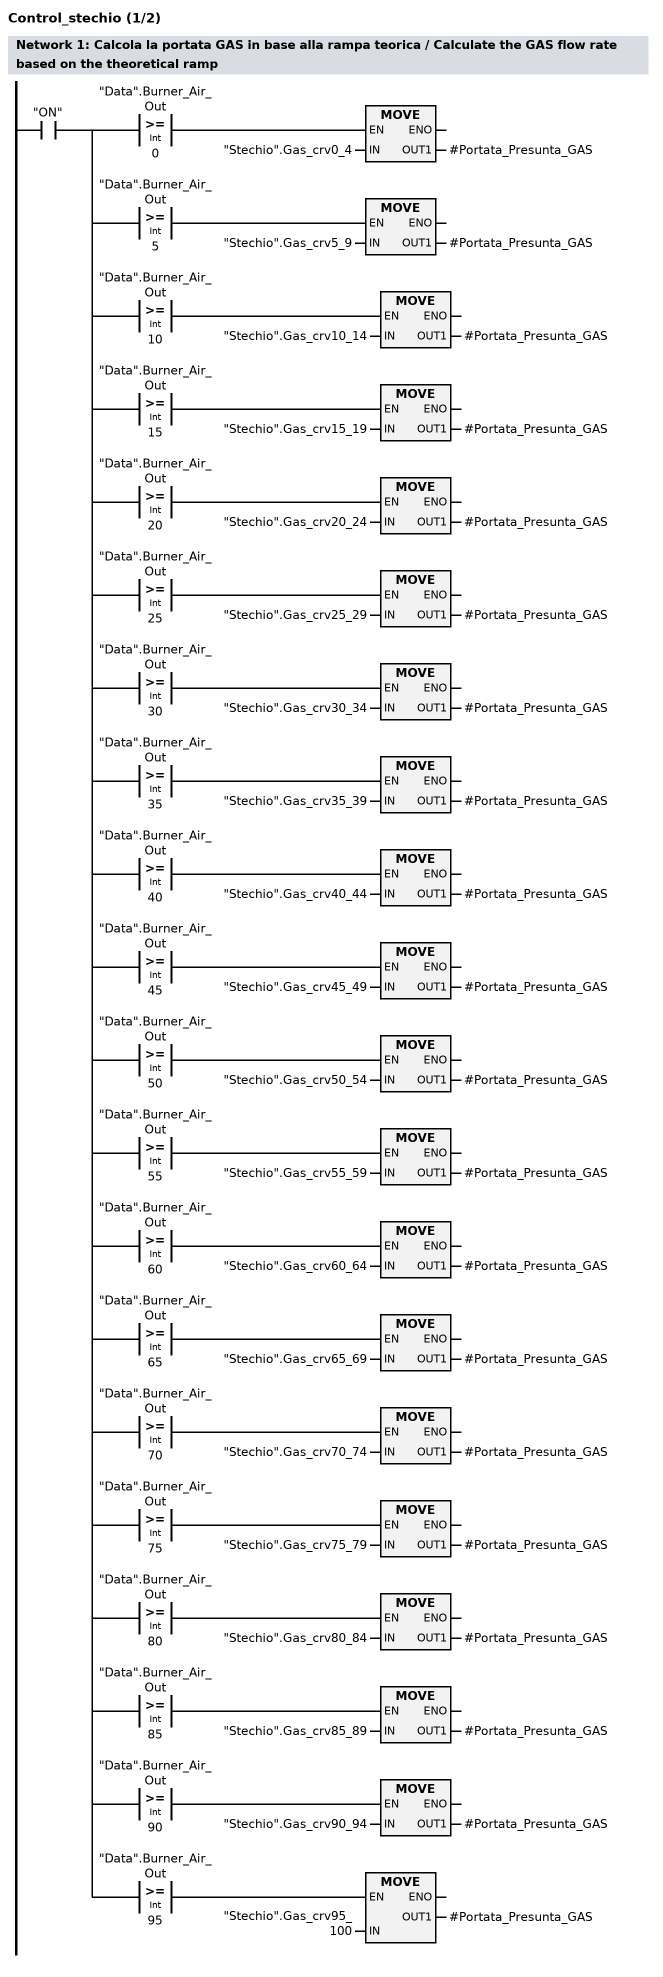
   RUNG wire#powerrail
      Contact( "ON" )
      wire#w1
      { S7_Templates := "SrcType := Int" } GE_Contact(in1 := "Data".Burner_Air_Out, in2 := 0)
      { S7_GenerateENO := "TRUE" } Move(in := "Stechio".Gas_crv0_4, out1 => #Portata_Presunta_GAS)
   END_RUNG
   RUNG wire#w1
      { S7_Templates := "SrcType := Int" } GE_Contact(in1 := "Data".Burner_Air_Out, in2 := 5)
      { S7_GenerateENO := "TRUE" } Move(in := "Stechio".Gas_crv5_9, out1 => #Portata_Presunta_GAS)
   END_RUNG
   RUNG wire#w1
      { S7_Templates := "SrcType := Int" } GE_Contact(in1 := "Data".Burner_Air_Out, in2 := 10)
      { S7_GenerateENO := "TRUE" } Move(in := "Stechio".Gas_crv10_14, out1 => #Portata_Presunta_GAS)
   END_RUNG
   RUNG wire#w1
      { S7_Templates := "SrcType := Int" } GE_Contact(in1 := "Data".Burner_Air_Out, in2 := 15)
      { S7_GenerateENO := "TRUE" } Move(in := "Stechio".Gas_crv15_19, out1 => #Portata_Presunta_GAS)
   END_RUNG
   RUNG wire#w1
      { S7_Templates := "SrcType := Int" } GE_Contact(in1 := "Data".Burner_Air_Out, in2 := 20)
      { S7_GenerateENO := "TRUE" } Move(in := "Stechio".Gas_crv20_24, out1 => #Portata_Presunta_GAS)
   END_RUNG
   RUNG wire#w1
      { S7_Templates := "SrcType := Int" } GE_Contact(in1 := "Data".Burner_Air_Out, in2 := 25)
      { S7_GenerateENO := "TRUE" } Move(in := "Stechio".Gas_crv25_29, out1 => #Portata_Presunta_GAS)
   END_RUNG
   RUNG wire#w1
      { S7_Templates := "SrcType := Int" } GE_Contact(in1 := "Data".Burner_Air_Out, in2 := 30)
      { S7_GenerateENO := "TRUE" } Move(in := "Stechio".Gas_crv30_34, out1 => #Portata_Presunta_GAS)
   END_RUNG
   RUNG wire#w1
      { S7_Templates := "SrcType := Int" } GE_Contact(in1 := "Data".Burner_Air_Out, in2 := 35)
      { S7_GenerateENO := "TRUE" } Move(in := "Stechio".Gas_crv35_39, out1 => #Portata_Presunta_GAS)
   END_RUNG
   RUNG wire#w1
      { S7_Templates := "SrcType := Int" } GE_Contact(in1 := "Data".Burner_Air_Out, in2 := 40)
      { S7_GenerateENO := "TRUE" } Move(in := "Stechio".Gas_crv40_44, out1 => #Portata_Presunta_GAS)
   END_RUNG
   RUNG wire#w1
      { S7_Templates := "SrcType := Int" } GE_Contact(in1 := "Data".Burner_Air_Out, in2 := 45)
      { S7_GenerateENO := "TRUE" } Move(in := "Stechio".Gas_crv45_49, out1 => #Portata_Presunta_GAS)
   END_RUNG
   RUNG wire#w1
      { S7_Templates := "SrcType := Int" } GE_Contact(in1 := "Data".Burner_Air_Out, in2 := 50)
      { S7_GenerateENO := "TRUE" } Move(in := "Stechio".Gas_crv50_54, out1 => #Portata_Presunta_GAS)
   END_RUNG
   RUNG wire#w1
      { S7_Templates := "SrcType := Int" } GE_Contact(in1 := "Data".Burner_Air_Out, in2 := 55)
      { S7_GenerateENO := "TRUE" } Move(in := "Stechio".Gas_crv55_59, out1 => #Portata_Presunta_GAS)
   END_RUNG
   RUNG wire#w1
      { S7_Templates := "SrcType := Int" } GE_Contact(in1 := "Data".Burner_Air_Out, in2 := 60)
      { S7_GenerateENO := "TRUE" } Move(in := "Stechio".Gas_crv60_64, out1 => #Portata_Presunta_GAS)
   END_RUNG
   RUNG wire#w1
      { S7_Templates := "SrcType := Int" } GE_Contact(in1 := "Data".Burner_Air_Out, in2 := 65)
      { S7_GenerateENO := "TRUE" } Move(in := "Stechio".Gas_crv65_69, out1 => #Portata_Presunta_GAS)
   END_RUNG
   RUNG wire#w1
      { S7_Templates := "SrcType := Int" } GE_Contact(in1 := "Data".Burner_Air_Out, in2 := 70)
      { S7_GenerateENO := "TRUE" } Move(in := "Stechio".Gas_crv70_74, out1 => #Portata_Presunta_GAS)
   END_RUNG
   RUNG wire#w1
      { S7_Templates := "SrcType := Int" } GE_Contact(in1 := "Data".Burner_Air_Out, in2 := 75)
      { S7_GenerateENO := "TRUE" } Move(in := "Stechio".Gas_crv75_79, out1 => #Portata_Presunta_GAS)
   END_RUNG
   RUNG wire#w1
      { S7_Templates := "SrcType := Int" } GE_Contact(in1 := "Data".Burner_Air_Out, in2 := 80)
      { S7_GenerateENO := "TRUE" } Move(in := "Stechio".Gas_crv80_84, out1 => #Portata_Presunta_GAS)
   END_RUNG
   RUNG wire#w1
      { S7_Templates := "SrcType := Int" } GE_Contact(in1 := "Data".Burner_Air_Out, in2 := 85)
      { S7_GenerateENO := "TRUE" } Move(in := "Stechio".Gas_crv85_89, out1 => #Portata_Presunta_GAS)
   END_RUNG
   RUNG wire#w1
      { S7_Templates := "SrcType := Int" } GE_Contact(in1 := "Data".Burner_Air_Out, in2 := 90)
      { S7_GenerateENO := "TRUE" } Move(in := "Stechio".Gas_crv90_94, out1 => #Portata_Presunta_GAS)
   END_RUNG
   RUNG wire#w1
      { S7_Templates := "SrcType := Int" } GE_Contact(in1 := "Data".Burner_Air_Out, in2 := 95)
      { S7_GenerateENO := "TRUE" } Move(in := "Stechio".Gas_crv95_100, out1 => #Portata_Presunta_GAS)
   END_RUNG
   // the same network as SCL:
   IF "ON" AND ("Data".Burner_Air_Out >= 0) THEN #Portata_Presunta_GAS := "Stechio".Gas_crv0_4; END_IF;
   IF "ON" AND ("Data".Burner_Air_Out >= 5) THEN #Portata_Presunta_GAS := "Stechio".Gas_crv5_9; END_IF;
   IF "ON" AND ("Data".Burner_Air_Out >= 10) THEN #Portata_Presunta_GAS := "Stechio".Gas_crv10_14; END_IF;
   IF "ON" AND ("Data".Burner_Air_Out >= 15) THEN #Portata_Presunta_GAS := "Stechio".Gas_crv15_19; END_IF;
   IF "ON" AND ("Data".Burner_Air_Out >= 20) THEN #Portata_Presunta_GAS := "Stechio".Gas_crv20_24; END_IF;
   IF "ON" AND ("Data".Burner_Air_Out >= 25) THEN #Portata_Presunta_GAS := "Stechio".Gas_crv25_29; END_IF;
   IF "ON" AND ("Data".Burner_Air_Out >= 30) THEN #Portata_Presunta_GAS := "Stechio".Gas_crv30_34; END_IF;
   IF "ON" AND ("Data".Burner_Air_Out >= 35) THEN #Portata_Presunta_GAS := "Stechio".Gas_crv35_39; END_IF;
   IF "ON" AND ("Data".Burner_Air_Out >= 40) THEN #Portata_Presunta_GAS := "Stechio".Gas_crv40_44; END_IF;
   IF "ON" AND ("Data".Burner_Air_Out >= 45) THEN #Portata_Presunta_GAS := "Stechio".Gas_crv45_49; END_IF;
   IF "ON" AND ("Data".Burner_Air_Out >= 50) THEN #Portata_Presunta_GAS := "Stechio".Gas_crv50_54; END_IF;
   IF "ON" AND ("Data".Burner_Air_Out >= 55) THEN #Portata_Presunta_GAS := "Stechio".Gas_crv55_59; END_IF;
   IF "ON" AND ("Data".Burner_Air_Out >= 60) THEN #Portata_Presunta_GAS := "Stechio".Gas_crv60_64; END_IF;
   IF "ON" AND ("Data".Burner_Air_Out >= 65) THEN #Portata_Presunta_GAS := "Stechio".Gas_crv65_69; END_IF;
   IF "ON" AND ("Data".Burner_Air_Out >= 70) THEN #Portata_Presunta_GAS := "Stechio".Gas_crv70_74; END_IF;
   IF "ON" AND ("Data".Burner_Air_Out >= 75) THEN #Portata_Presunta_GAS := "Stechio".Gas_crv75_79; END_IF;
   IF "ON" AND ("Data".Burner_Air_Out >= 80) THEN #Portata_Presunta_GAS := "Stechio".Gas_crv80_84; END_IF;
   IF "ON" AND ("Data".Burner_Air_Out >= 85) THEN #Portata_Presunta_GAS := "Stechio".Gas_crv85_89; END_IF;
   IF "ON" AND ("Data".Burner_Air_Out >= 90) THEN #Portata_Presunta_GAS := "Stechio".Gas_crv90_94; END_IF;
   IF "ON" AND ("Data".Burner_Air_Out >= 95) THEN #Portata_Presunta_GAS := "Stechio".Gas_crv95_100; END_IF;
END_REGION

REGION Network 2 (STL): Calcolo del rapporto stechiometrico attuale / Calculation of the current stoichiometric ratio

         L     "Data".MASSICO_FLOW_AIR;  //Converte portata aria
         ITD;
         DTR;
         T     #AIR_FLOW;  //In reale



         L     "Data".MASSICO_FLOW_GAS;  //Converte portata gas
         ITD;
         DTR;
         T     #GAS_FLOW;  //In reale


   //------------------------------------------------------------------------

         L     #AIR_FLOW;  //Calcola il rapporto
         L     #GAS_FLOW;  //Stechiometrico
         /R;
         T     #Stechio_attuale;  //(portata aria) / (portata gas)

         L     #Stechio_attuale;
         T     "Stechio".Real_stechio;  //(portata aria) / (portata gas)


         L     "Stechio".Set_stechio;
         T     #SetPoint_Stechio;

   //------------------------------------------------------------------------
END_REGION

REGION Network 3: Esegue blocco PID / Run PID block
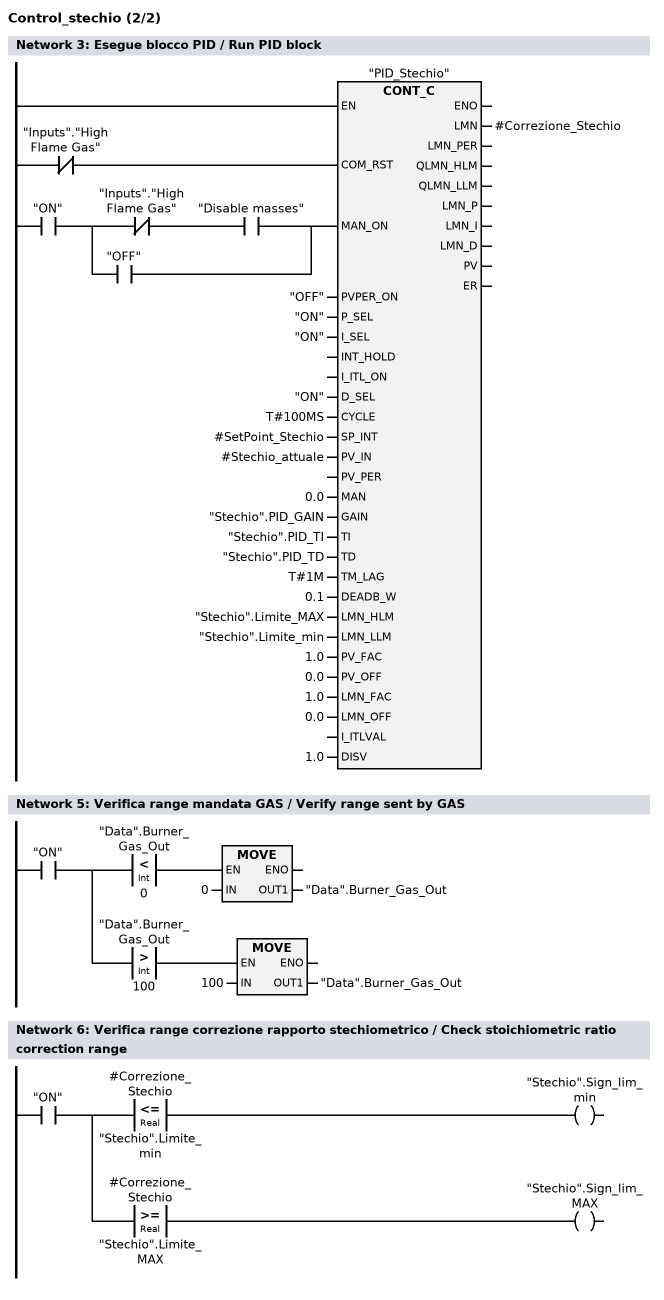
   "PID_Stechio"(COM_RST := NOT "Inputs"."High Flame Gas",   // CONT_C
                 MAN_ON := "ON" AND ((NOT "Inputs"."High Flame Gas" AND "Disable masses") OR "OFF"),
                 PVPER_ON := "OFF",
                 P_SEL := "ON",
                 I_SEL := "ON",
                 D_SEL := "ON",
                 CYCLE := T#100MS,
                 SP_INT := #SetPoint_Stechio,
                 PV_IN := #Stechio_attuale,
                 MAN := 0.0,
                 GAIN := "Stechio".PID_GAIN,
                 TI := "Stechio".PID_TI,
                 TD := "Stechio".PID_TD,
                 TM_LAG := T#1M,
                 DEADB_W := 0.1,
                 LMN_HLM := "Stechio".Limite_MAX,
                 LMN_LLM := "Stechio".Limite_min,
                 PV_FAC := 1.0,
                 PV_OFF := 0.0,
                 LMN_FAC := 1.0,
                 LMN_OFF := 0.0,
                 DISV := 1.0,
                 LMN => #Correzione_Stechio);
END_REGION

REGION Network 4 (STL): Calcolo percentuale gas ed invia / Calculate percentage and send
   //Converte Correzione calcolata in intero
         L     #Correzione_Stechio;
         RND;
         T     #Correzione_Calcolata_INT;


   //e corregge la portata del GAS
   //portata GAS = portata presunta gas + correzione stechiometrica

         L     #Portata_Presunta_GAS;
         L     #Correzione_Calcolata_INT;
         +I;

         T     "Data".Burner_Gas_Out;
END_REGION

REGION Network 5: Verifica range mandata GAS / Verify range sent by GAS
   RUNG wire#powerrail
      Contact( "ON" )
      wire#w1
      { S7_Templates := "SrcType := Int" } LT_Contact(in1 := "Data".Burner_Gas_Out, in2 := 0)
      { S7_GenerateENO := "TRUE" } Move(in := 0, out1 => "Data".Burner_Gas_Out)
   END_RUNG
   RUNG wire#w1
      { S7_Templates := "SrcType := Int" } GT_Contact(in1 := "Data".Burner_Gas_Out, in2 := 100)
      { S7_GenerateENO := "TRUE" } Move(in := 100, out1 => "Data".Burner_Gas_Out)
   END_RUNG
   // the same network as SCL:
   IF "ON" AND ("Data".Burner_Gas_Out < 0) THEN "Data".Burner_Gas_Out := 0; END_IF;
   IF "ON" AND ("Data".Burner_Gas_Out > 100) THEN "Data".Burner_Gas_Out := 100; END_IF;
END_REGION

REGION Network 6: Verifica range correzione rapporto stechiometrico / Check stoichiometric ratio correction range
   RUNG wire#powerrail
      Contact( "ON" )
      wire#w1
      { S7_Templates := "SrcType := Real" } LE_Contact(in1 := #Correzione_Stechio, in2 := "Stechio".Limite_min)
      Coil( "Stechio".Sign_lim_min )
   END_RUNG
   RUNG wire#w1
      { S7_Templates := "SrcType := Real" } GE_Contact(in1 := #Correzione_Stechio, in2 := "Stechio".Limite_MAX)
      Coil( "Stechio".Sign_lim_MAX )
   END_RUNG
   // the same network as SCL:
   "Stechio".Sign_lim_min := "ON" AND (#Correzione_Stechio <= "Stechio".Limite_min);
   "Stechio".Sign_lim_MAX := "ON" AND (#Correzione_Stechio >= "Stechio".Limite_MAX);
END_REGION

REGION Network 7 (STL): Contatore metri cubi gas passati / Meter of cubic meters of gas passed
   //------------------------------------------------------------------------
   //Calcolo consumo GAS test
   //------------------------------------------------------------------------


         AN    "Inputs"."Burner On";
         JC    FINE;

         L     #GAS_FLOW;
         L     36000.0;
         /R;
         T     #Portata_al_secondo;

         L     #Portata_al_secondo;
         L     "Stechio".Consumo_GAS;
         +R;
         T     "Stechio".Consumo_GAS;

         L     #Portata_al_secondo;
         L     "Stechio".Consumo_GAS_TOTALE;
         +R;
         T     "Stechio".Consumo_GAS_TOTALE;

         JU    FINE;

   AZZ:  L     0;
         T     "Stechio".Consumo_GAS;
   FINE: NOP   0;
   //------------------------------------------------------------------------

         AN    "HMI_DB".ResetCounter_GasConsumption;
         JC    azz0;
         L     0;
         T     "Stechio".Consumo_GAS;
         SET;
         R     "HMI_DB".ResetCounter_GasConsumption;
   azz0: NOP   0;
END_REGION
END_FUNCTION

FUNCTION "Valve Control loop" : Void   // FC14, LAD
TITLE = Motorized valves loop control
{ S7_Optimized_Access := 'FALSE' }
VERSION : 0.1
   VAR_TEMP
      App00 : S5Time;
      App01 : S5Time;
      App02 : S5Time;
      App03 : S5Time;
      App04 : Int;
      App05 : S5Time;
      App6 : Int;
      AppVG01 : Int;
      ErrPSH02 : Int;
      ErrPSH03 : Int;
   END_VAR
   VAR_TEMP   // added for the SCL form of the ladder/FBD networks
      _w1 : Bool;
      _w2 : Bool;
      _w3 : Bool;
      _w4 : Bool;
      _w5 : Bool;
      _w6 : Bool;
      _w7 : Bool;
      _w8 : Bool;
   END_VAR
BEGIN

REGION Network 1: MV01 Controlled by TC03
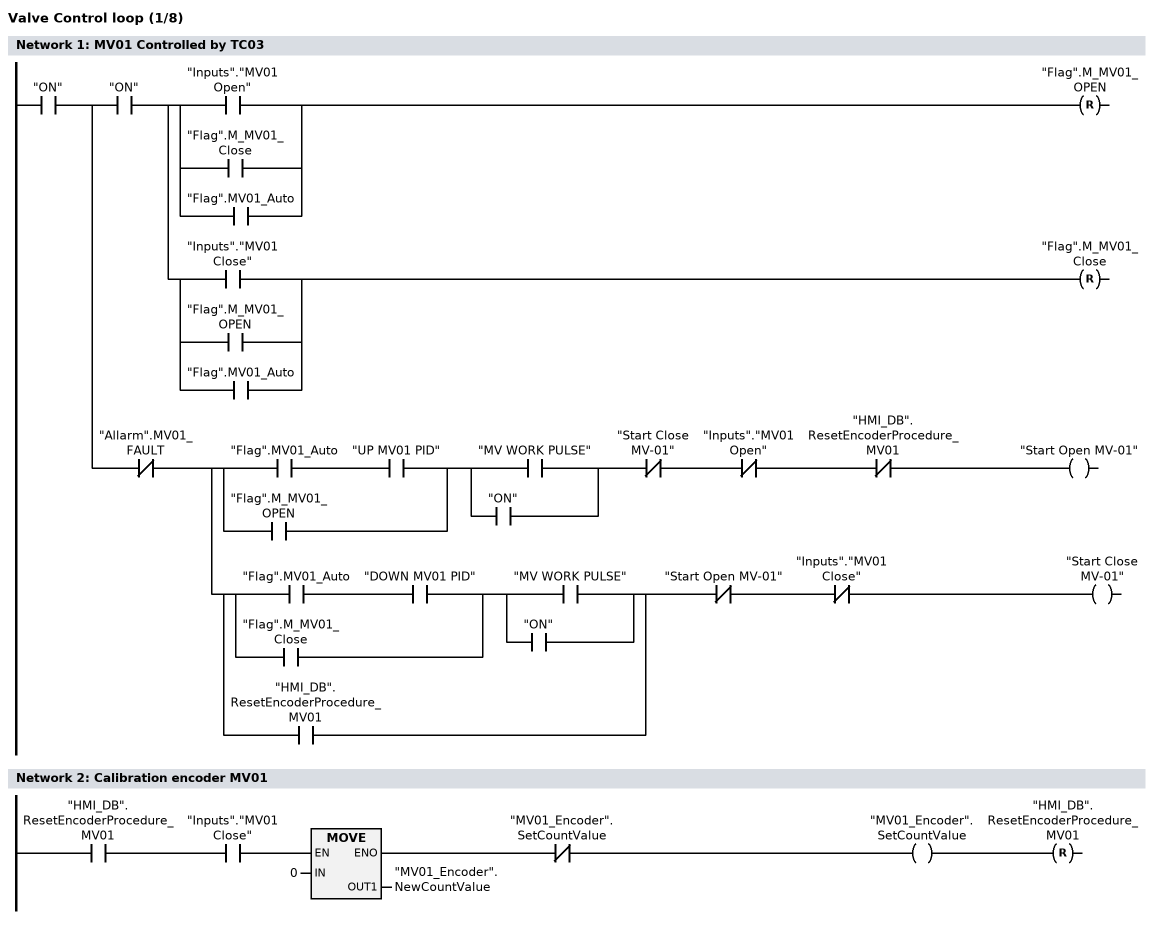
   RUNG wire#powerrail
      Contact( "ON" )
      wire#w1
      Contact( "ON" )
      wire#w2
      Contact( "Inputs"."MV01 Open" )
      wire#w3
      R_Coil( "Flag".M_MV01_OPEN )
   END_RUNG
   RUNG wire#w2
      Contact( "Flag".M_MV01_Close )
   END_RUNG wire#w3
   RUNG wire#w2
      Contact( "Flag".MV01_Auto )
   END_RUNG wire#w3
   RUNG wire#w2
      Contact( "Inputs"."MV01 Close" )
      wire#w4
      R_Coil( "Flag".M_MV01_Close )
   END_RUNG
   RUNG wire#w2
      Contact( "Flag".M_MV01_OPEN )
   END_RUNG wire#w4
   RUNG wire#w2
      Contact( "Flag".MV01_Auto )
   END_RUNG wire#w4
   RUNG wire#w1
      I_Contact( "Allarm".MV01_FAULT )
      wire#w5
      Contact( "Flag".MV01_Auto )
      Contact( "UP MV01 PID" )
      wire#w6
      Contact( "MV WORK PULSE" )
      wire#w7
      I_Contact( "Start Close MV-01" )
      I_Contact( "Inputs"."MV01 Open" )
      I_Contact( "HMI_DB".ResetEncoderProcedure_MV01 )
      Coil( "Start Open MV-01" )
   END_RUNG
   RUNG wire#w5
      Contact( "Flag".M_MV01_OPEN )
   END_RUNG wire#w6
   RUNG wire#w6
      Contact( "ON" )
   END_RUNG wire#w7
   RUNG wire#w5
      Contact( "Flag".MV01_Auto )
      Contact( "DOWN MV01 PID" )
      wire#w8
      Contact( "MV WORK PULSE" )
      wire#w9
      I_Contact( "Start Open MV-01" )
      I_Contact( "Inputs"."MV01 Close" )
      Coil( "Start Close MV-01" )
   END_RUNG
   RUNG wire#w5
      Contact( "Flag".M_MV01_Close )
   END_RUNG wire#w8
   RUNG wire#w8
      Contact( "ON" )
   END_RUNG wire#w9
   RUNG wire#w5
      Contact( "HMI_DB".ResetEncoderProcedure_MV01 )
   END_RUNG wire#w9
   // the same network as SCL:
   #_w1 := "ON" AND "ON";
   IF #_w1 AND ("Inputs"."MV01 Open" OR "Flag".M_MV01_Close OR "Flag".MV01_Auto) THEN
       "Flag".M_MV01_OPEN := FALSE;
   END_IF;
   IF #_w1 AND ("Inputs"."MV01 Close" OR "Flag".M_MV01_OPEN OR "Flag".MV01_Auto) THEN
       "Flag".M_MV01_Close := FALSE;
   END_IF;
   #_w2 := "ON" AND NOT "Allarm".MV01_FAULT;
   "Start Open MV-01" := #_w2 AND (("Flag".MV01_Auto AND "UP MV01 PID") OR "Flag".M_MV01_OPEN) AND ("MV WORK PULSE" OR "ON") AND NOT "Start Close MV-01" AND NOT "Inputs"."MV01 Open" AND NOT "HMI_DB".ResetEncoderProcedure_MV01;
   "Start Close MV-01" := #_w2 AND (((("Flag".MV01_Auto AND "DOWN MV01 PID") OR "Flag".M_MV01_Close) AND ("MV WORK PULSE" OR "ON")) OR "HMI_DB".ResetEncoderProcedure_MV01) AND NOT "Start Open MV-01" AND NOT "Inputs"."MV01 Close";
END_REGION

REGION Network 2: Calibration encoder MV01
   RUNG wire#powerrail
      Contact( "HMI_DB".ResetEncoderProcedure_MV01 )
      Contact( "Inputs"."MV01 Close" )
      Move(in := 0, out1 => "MV01_Encoder".NewCountValue)
      I_Contact( "MV01_Encoder".SetCountValue )
      Coil( "MV01_Encoder".SetCountValue )
      R_Coil( "HMI_DB".ResetEncoderProcedure_MV01 )
   END_RUNG
   // the same network as SCL:
   #_w1 := "HMI_DB".ResetEncoderProcedure_MV01 AND "Inputs"."MV01 Close";
   IF #_w1 THEN "MV01_Encoder".NewCountValue := 0; END_IF;
   "MV01_Encoder".SetCountValue := #_w1 AND NOT "MV01_Encoder".SetCountValue;
   IF "MV01_Encoder".SetCountValue THEN "HMI_DB".ResetEncoderProcedure_MV01 := FALSE; END_IF;
END_REGION

REGION Network 3: MV02 Controlled by PSH-01
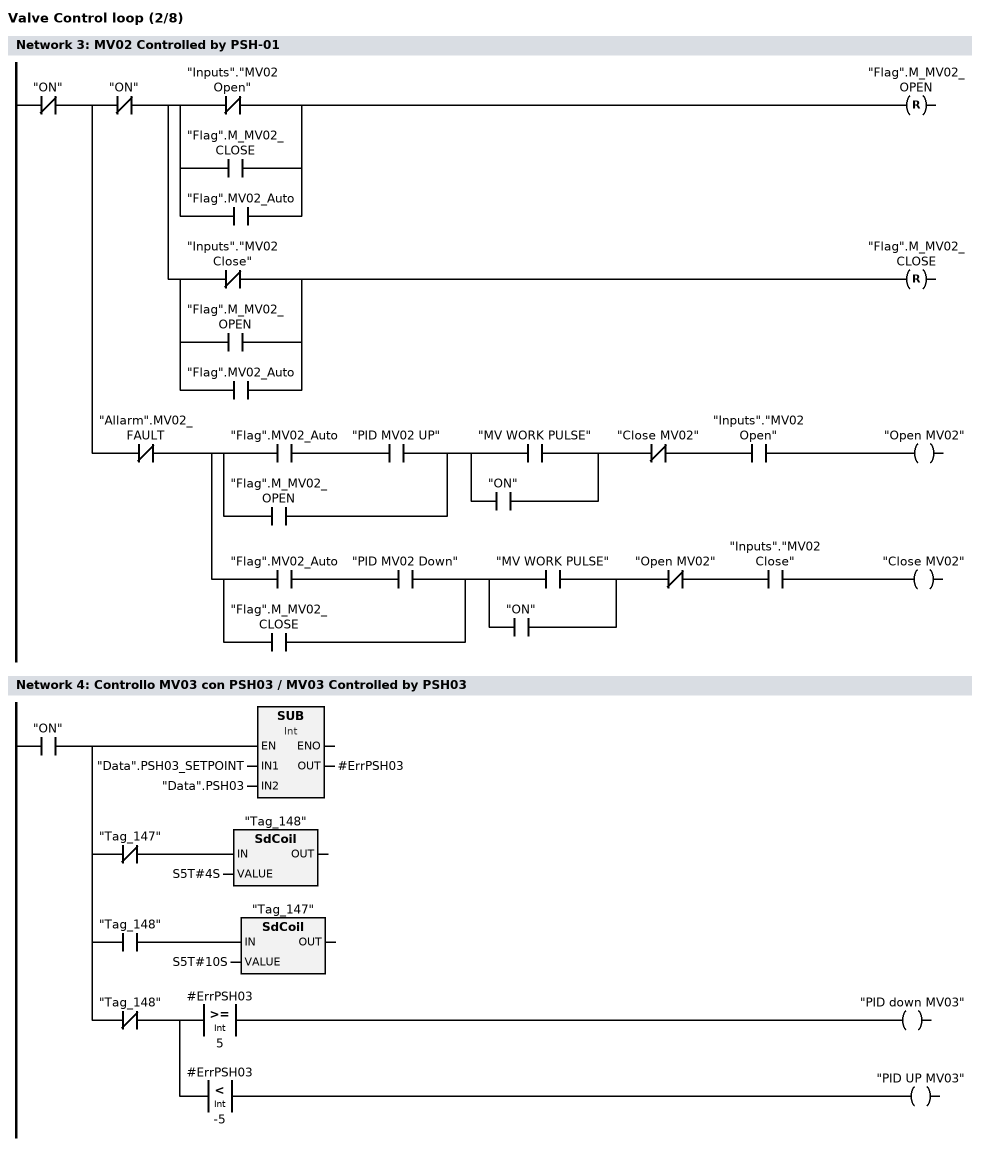
   RUNG wire#powerrail
      I_Contact( "ON" )
      wire#w1
      I_Contact( "ON" )
      wire#w2
      I_Contact( "Inputs"."MV02 Open" )
      wire#w3
      R_Coil( "Flag".M_MV02_OPEN )
   END_RUNG
   RUNG wire#w2
      Contact( "Flag".M_MV02_CLOSE )
   END_RUNG wire#w3
   RUNG wire#w2
      Contact( "Flag".MV02_Auto )
   END_RUNG wire#w3
   RUNG wire#w2
      I_Contact( "Inputs"."MV02 Close" )
      wire#w4
      R_Coil( "Flag".M_MV02_CLOSE )
   END_RUNG
   RUNG wire#w2
      Contact( "Flag".M_MV02_OPEN )
   END_RUNG wire#w4
   RUNG wire#w2
      Contact( "Flag".MV02_Auto )
   END_RUNG wire#w4
   RUNG wire#w1
      I_Contact( "Allarm".MV02_FAULT )
      wire#w5
      Contact( "Flag".MV02_Auto )
      Contact( "PID MV02 UP" )
      wire#w6
      Contact( "MV WORK PULSE" )
      wire#w7
      I_Contact( "Close MV02" )
      Contact( "Inputs"."MV02 Open" )
      Coil( "Open MV02" )
   END_RUNG
   RUNG wire#w5
      Contact( "Flag".M_MV02_OPEN )
   END_RUNG wire#w6
   RUNG wire#w6
      Contact( "ON" )
   END_RUNG wire#w7
   RUNG wire#w5
      Contact( "Flag".MV02_Auto )
      Contact( "PID MV02 Down" )
      wire#w8
      Contact( "MV WORK PULSE" )
      wire#w9
      I_Contact( "Open MV02" )
      Contact( "Inputs"."MV02 Close" )
      Coil( "Close MV02" )
   END_RUNG
   RUNG wire#w5
      Contact( "Flag".M_MV02_CLOSE )
   END_RUNG wire#w8
   RUNG wire#w8
      Contact( "ON" )
   END_RUNG wire#w9
   // the same network as SCL:
   #_w1 := NOT "ON" AND NOT "ON";
   IF #_w1 AND (NOT "Inputs"."MV02 Open" OR "Flag".M_MV02_CLOSE OR "Flag".MV02_Auto) THEN
       "Flag".M_MV02_OPEN := FALSE;
   END_IF;
   IF #_w1 AND (NOT "Inputs"."MV02 Close" OR "Flag".M_MV02_OPEN OR "Flag".MV02_Auto) THEN
       "Flag".M_MV02_CLOSE := FALSE;
   END_IF;
   #_w2 := NOT "ON" AND NOT "Allarm".MV02_FAULT;
   "Open MV02" := #_w2 AND (("Flag".MV02_Auto AND "PID MV02 UP") OR "Flag".M_MV02_OPEN) AND ("MV WORK PULSE" OR "ON") AND NOT "Close MV02" AND "Inputs"."MV02 Open";
   "Close MV02" := #_w2 AND (("Flag".MV02_Auto AND "PID MV02 Down") OR "Flag".M_MV02_CLOSE) AND ("MV WORK PULSE" OR "ON") AND NOT "Open MV02" AND "Inputs"."MV02 Close";
END_REGION

REGION Network 4: Controllo MV03 con PSH03 / MV03 Controlled by PSH03
   // no SCL statement known for SdCoil: written as a call
   IF "ON" THEN #ErrPSH03 := "Data".PSH03_SETPOINT - "Data".PSH03; END_IF;
   #_w1 := "ON";
   SdCoil(in := "ON" AND NOT "Tag_147", value := S5T#4S, operand := "Tag_148");
   SdCoil(in := #_w1 AND "Tag_148", value := S5T#10S, operand := "Tag_147");
   #_w2 := #_w1 AND NOT "Tag_148";
   "PID down MV03" := #_w2 AND (#ErrPSH03 >= 5);
   "PID UP MV03" := #_w2 AND (#ErrPSH03 < (-5));
END_REGION

REGION Network 5: MV03 Controlled by PSH03
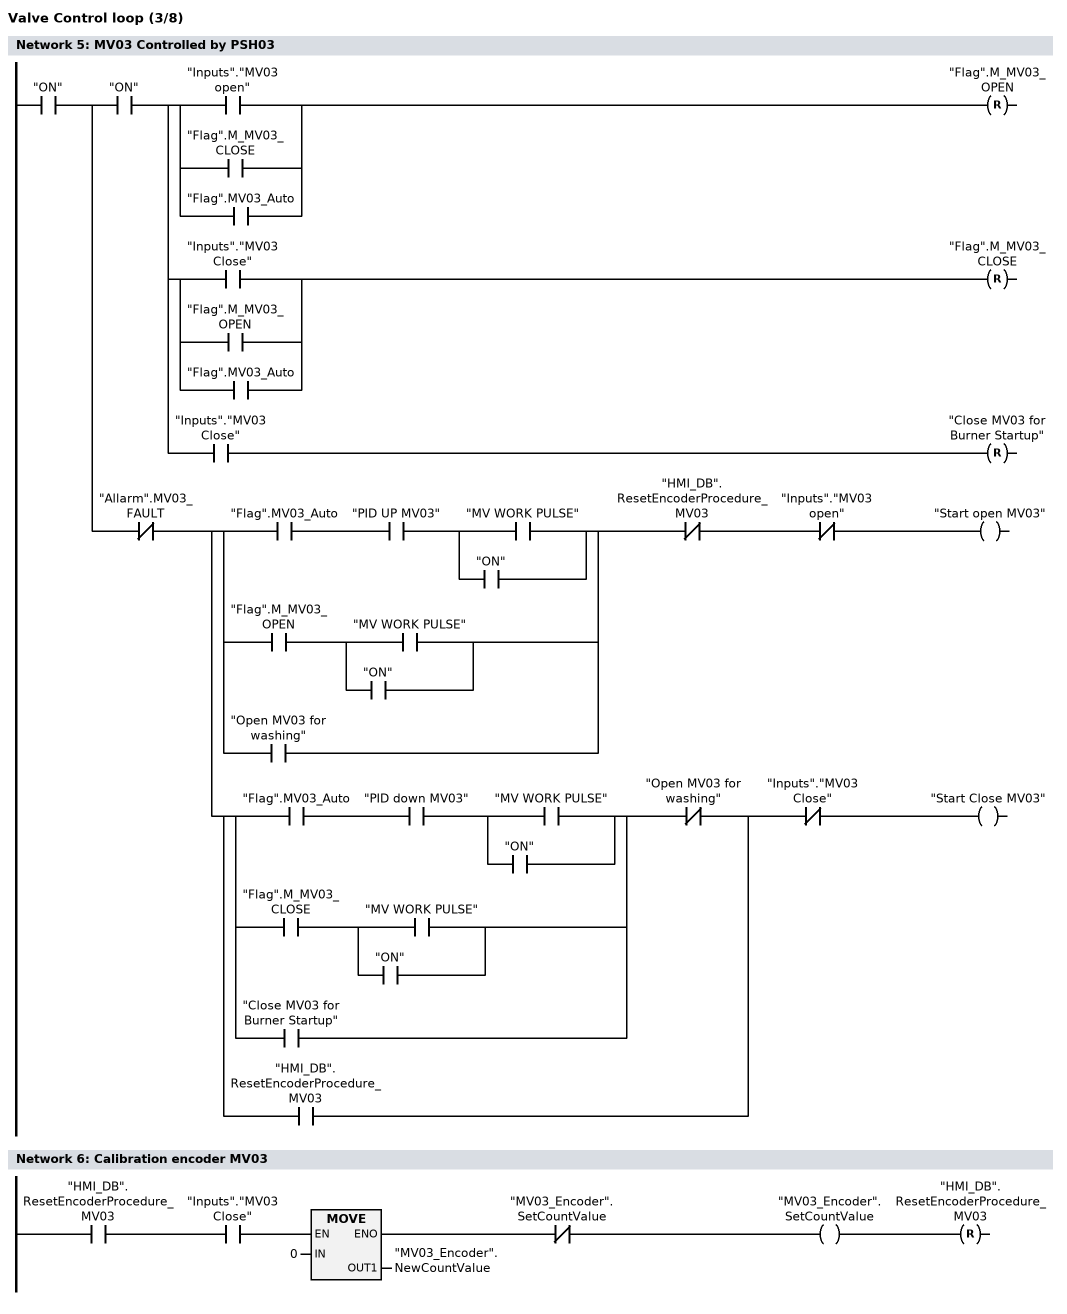
   RUNG wire#powerrail
      Contact( "ON" )
      wire#w1
      Contact( "ON" )
      wire#w2
      Contact( "Inputs"."MV03 open" )
      wire#w3
      R_Coil( "Flag".M_MV03_OPEN )
   END_RUNG
   RUNG wire#w2
      Contact( "Flag".M_MV03_CLOSE )
   END_RUNG wire#w3
   RUNG wire#w2
      Contact( "Flag".MV03_Auto )
   END_RUNG wire#w3
   RUNG wire#w2
      Contact( "Inputs"."MV03 Close" )
      wire#w4
      R_Coil( "Flag".M_MV03_CLOSE )
   END_RUNG
   RUNG wire#w2
      Contact( "Flag".M_MV03_OPEN )
   END_RUNG wire#w4
   RUNG wire#w2
      Contact( "Flag".MV03_Auto )
   END_RUNG wire#w4
   RUNG wire#w2
      Contact( "Inputs"."MV03 Close" )
      R_Coil( "Close MV03 for Burner Startup" )
   END_RUNG
   RUNG wire#w1
      I_Contact( "Allarm".MV03_FAULT )
      wire#w5
      Contact( "Flag".MV03_Auto )
      Contact( "PID UP MV03" )
      wire#w6
      Contact( "MV WORK PULSE" )
      wire#w7
      I_Contact( "HMI_DB".ResetEncoderProcedure_MV03 )
      I_Contact( "Inputs"."MV03 open" )
      Coil( "Start open MV03" )
   END_RUNG
   RUNG wire#w6
      Contact( "ON" )
   END_RUNG wire#w7
   RUNG wire#w5
      Contact( "Flag".M_MV03_OPEN )
      wire#w8
      Contact( "MV WORK PULSE" )
   END_RUNG wire#w7
   RUNG wire#w8
      Contact( "ON" )
   END_RUNG wire#w7
   RUNG wire#w5
      Contact( "Open MV03 for washing" )
   END_RUNG wire#w7
   RUNG wire#w5
      Contact( "Flag".MV03_Auto )
      Contact( "PID down MV03" )
      wire#w9
      Contact( "MV WORK PULSE" )
      wire#w10
      I_Contact( "Open MV03 for washing" )
      wire#w12
      I_Contact( "Inputs"."MV03 Close" )
      Coil( "Start Close MV03" )
   END_RUNG
   RUNG wire#w9
      Contact( "ON" )
   END_RUNG wire#w10
   RUNG wire#w5
      Contact( "Flag".M_MV03_CLOSE )
      wire#w11
      Contact( "MV WORK PULSE" )
   END_RUNG wire#w10
   RUNG wire#w11
      Contact( "ON" )
   END_RUNG wire#w10
   RUNG wire#w5
      Contact( "Close MV03 for Burner Startup" )
   END_RUNG wire#w10
   RUNG wire#w5
      Contact( "HMI_DB".ResetEncoderProcedure_MV03 )
   END_RUNG wire#w12
   // the same network as SCL:
   #_w1 := "ON" AND "ON";
   IF #_w1 AND ("Inputs"."MV03 open" OR "Flag".M_MV03_CLOSE OR "Flag".MV03_Auto) THEN
       "Flag".M_MV03_OPEN := FALSE;
   END_IF;
   IF #_w1 AND ("Inputs"."MV03 Close" OR "Flag".M_MV03_OPEN OR "Flag".MV03_Auto) THEN
       "Flag".M_MV03_CLOSE := FALSE;
   END_IF;
   IF #_w1 AND "Inputs"."MV03 Close" THEN "Close MV03 for Burner Startup" := FALSE; END_IF;
   #_w2 := "ON" AND NOT "Allarm".MV03_FAULT;
   "Start open MV03" := #_w2 AND (("Flag".MV03_Auto AND "PID UP MV03" AND ("MV WORK PULSE" OR "ON")) OR ("Flag".M_MV03_OPEN AND ("MV WORK PULSE" OR "ON")) OR "Open MV03 for washing") AND NOT "HMI_DB".ResetEncoderProcedure_MV03 AND NOT "Inputs"."MV03 open";
   "Start Close MV03" := #_w2 AND (((("Flag".MV03_Auto AND "PID down MV03" AND ("MV WORK PULSE" OR "ON")) OR ("Flag".M_MV03_CLOSE AND ("MV WORK PULSE" OR "ON")) OR "Close MV03 for Burner Startup") AND NOT "Open MV03 for washing") OR "HMI_DB".ResetEncoderProcedure_MV03) AND NOT "Inputs"."MV03 Close";
END_REGION

REGION Network 6: Calibration encoder MV03
   RUNG wire#powerrail
      Contact( "HMI_DB".ResetEncoderProcedure_MV03 )
      Contact( "Inputs"."MV03 Close" )
      Move(in := 0, out1 => "MV03_Encoder".NewCountValue)
      I_Contact( "MV03_Encoder".SetCountValue )
      Coil( "MV03_Encoder".SetCountValue )
      R_Coil( "HMI_DB".ResetEncoderProcedure_MV03 )
   END_RUNG
   // the same network as SCL:
   #_w1 := "HMI_DB".ResetEncoderProcedure_MV03 AND "Inputs"."MV03 Close";
   IF #_w1 THEN "MV03_Encoder".NewCountValue := 0; END_IF;
   "MV03_Encoder".SetCountValue := #_w1 AND NOT "MV03_Encoder".SetCountValue;
   IF "MV03_Encoder".SetCountValue THEN "HMI_DB".ResetEncoderProcedure_MV03 := FALSE; END_IF;
END_REGION

REGION Network 7: MV05 Controlled by RO-01
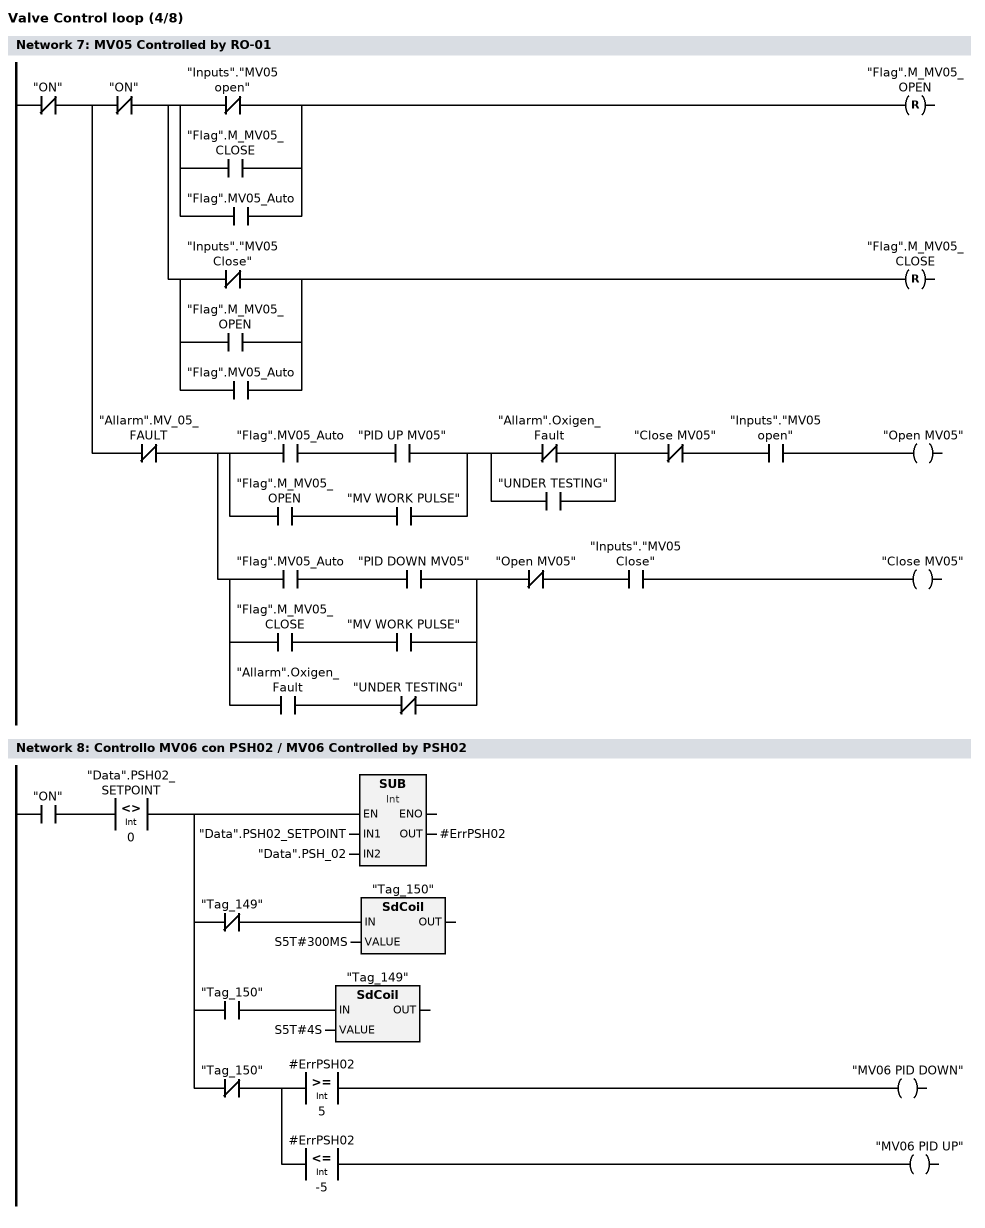
   RUNG wire#powerrail
      I_Contact( "ON" )
      wire#w1
      I_Contact( "ON" )
      wire#w2
      I_Contact( "Inputs"."MV05 open" )
      wire#w3
      R_Coil( "Flag".M_MV05_OPEN )
   END_RUNG
   RUNG wire#w2
      Contact( "Flag".M_MV05_CLOSE )
   END_RUNG wire#w3
   RUNG wire#w2
      Contact( "Flag".MV05_Auto )
   END_RUNG wire#w3
   RUNG wire#w2
      I_Contact( "Inputs"."MV05 Close" )
      wire#w4
      R_Coil( "Flag".M_MV05_CLOSE )
   END_RUNG
   RUNG wire#w2
      Contact( "Flag".M_MV05_OPEN )
   END_RUNG wire#w4
   RUNG wire#w2
      Contact( "Flag".MV05_Auto )
   END_RUNG wire#w4
   RUNG wire#w1
      I_Contact( "Allarm".MV_05_FAULT )
      wire#w5
      Contact( "Flag".MV05_Auto )
      Contact( "PID UP MV05" )
      wire#w6
      I_Contact( "Allarm".Oxigen_Fault )
      wire#w7
      I_Contact( "Close MV05" )
      Contact( "Inputs"."MV05 open" )
      Coil( "Open MV05" )
   END_RUNG
   RUNG wire#w5
      Contact( "Flag".M_MV05_OPEN )
      Contact( "MV WORK PULSE" )
   END_RUNG wire#w6
   RUNG wire#w6
      Contact( "UNDER TESTING" )
   END_RUNG wire#w7
   RUNG wire#w5
      Contact( "Flag".MV05_Auto )
      Contact( "PID DOWN MV05" )
      wire#w8
      I_Contact( "Open MV05" )
      Contact( "Inputs"."MV05 Close" )
      Coil( "Close MV05" )
   END_RUNG
   RUNG wire#w5
      Contact( "Flag".M_MV05_CLOSE )
      Contact( "MV WORK PULSE" )
   END_RUNG wire#w8
   RUNG wire#w5
      Contact( "Allarm".Oxigen_Fault )
      I_Contact( "UNDER TESTING" )
   END_RUNG wire#w8
   // the same network as SCL:
   #_w1 := NOT "ON" AND NOT "ON";
   IF #_w1 AND (NOT "Inputs"."MV05 open" OR "Flag".M_MV05_CLOSE OR "Flag".MV05_Auto) THEN
       "Flag".M_MV05_OPEN := FALSE;
   END_IF;
   IF #_w1 AND (NOT "Inputs"."MV05 Close" OR "Flag".M_MV05_OPEN OR "Flag".MV05_Auto) THEN
       "Flag".M_MV05_CLOSE := FALSE;
   END_IF;
   #_w2 := NOT "ON" AND NOT "Allarm".MV_05_FAULT;
   "Open MV05" := #_w2 AND (("Flag".MV05_Auto AND "PID UP MV05") OR ("Flag".M_MV05_OPEN AND "MV WORK PULSE")) AND (NOT "Allarm".Oxigen_Fault OR "UNDER TESTING") AND NOT "Close MV05" AND "Inputs"."MV05 open";
   "Close MV05" := #_w2 AND (("Flag".MV05_Auto AND "PID DOWN MV05") OR ("Flag".M_MV05_CLOSE AND "MV WORK PULSE") OR ("Allarm".Oxigen_Fault AND NOT "UNDER TESTING")) AND NOT "Open MV05" AND "Inputs"."MV05 Close";
END_REGION

REGION Network 8: Controllo MV06 con PSH02 / MV06 Controlled by PSH02
   // no SCL statement known for SdCoil: written as a call
   #_w1 := "ON" AND ("Data".PSH02_SETPOINT <> 0);
   IF #_w1 THEN #ErrPSH02 := "Data".PSH02_SETPOINT - "Data".PSH_02; END_IF;
   SdCoil(in := #_w1 AND NOT "Tag_149", value := S5T#300MS, operand := "Tag_150");
   SdCoil(in := #_w1 AND "Tag_150", value := S5T#4S, operand := "Tag_149");
   #_w2 := #_w1 AND NOT "Tag_150";
   "MV06 PID DOWN" := #_w2 AND (#ErrPSH02 >= 5);
   "MV06 PID UP" := #_w2 AND (#ErrPSH02 <= (-5));
END_REGION

REGION Network 9: Lo strumento ha un range di lavoro molto basso / The working tool has a low range
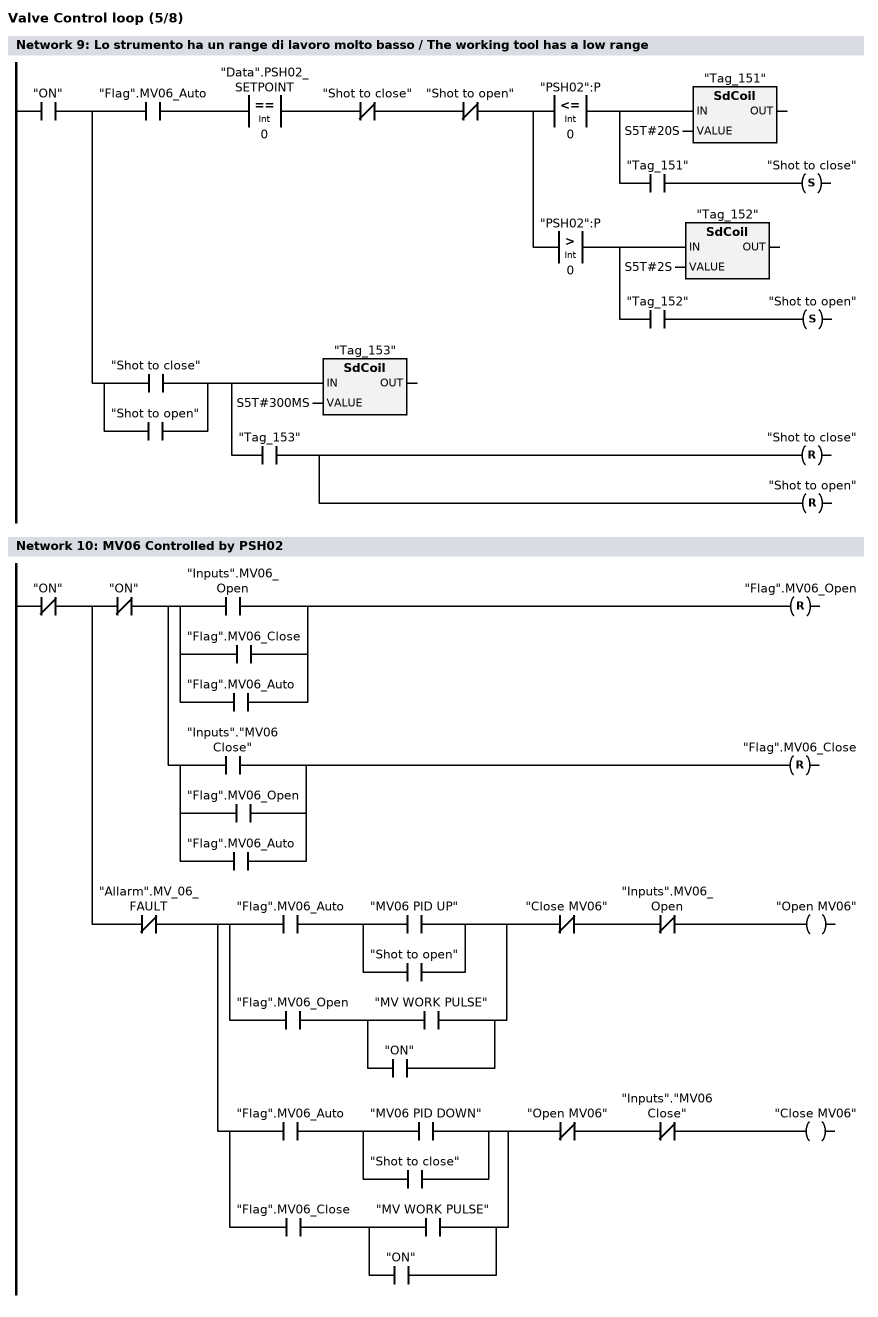
   // no SCL statement known for SdCoil: written as a call
   #_w1 := "ON" AND "Flag".MV06_Auto AND ("Data".PSH02_SETPOINT = 0) AND NOT "Shot to close" AND NOT "Shot to open";
   #_w2 := #_w1 AND ("PSH02":P <= 0);
   #_w3 := "ON";
   SdCoil(in := #_w2, value := S5T#20S, operand := "Tag_151");
   IF #_w2 AND "Tag_151" THEN "Shot to close" := TRUE; END_IF;
   #_w4 := #_w1 AND ("PSH02":P > 0);
   SdCoil(in := #_w4, value := S5T#2S, operand := "Tag_152");
   IF #_w4 AND "Tag_152" THEN "Shot to open" := TRUE; END_IF;
   #_w5 := #_w3 AND ("Shot to close" OR "Shot to open");
   SdCoil(in := #_w5, value := S5T#300MS, operand := "Tag_153");
   IF #_w5 AND "Tag_153" THEN
       "Shot to close" := FALSE;
       "Shot to open" := FALSE;
   END_IF;
END_REGION

REGION Network 10: MV06 Controlled by PSH02
   RUNG wire#powerrail
      I_Contact( "ON" )
      wire#w1
      I_Contact( "ON" )
      wire#w2
      Contact( "Inputs".MV06_Open )
      wire#w3
      R_Coil( "Flag".MV06_Open )
   END_RUNG
   RUNG wire#w2
      Contact( "Flag".MV06_Close )
   END_RUNG wire#w3
   RUNG wire#w2
      Contact( "Flag".MV06_Auto )
   END_RUNG wire#w3
   RUNG wire#w2
      Contact( "Inputs"."MV06 Close" )
      wire#w4
      R_Coil( "Flag".MV06_Close )
   END_RUNG
   RUNG wire#w2
      Contact( "Flag".MV06_Open )
   END_RUNG wire#w4
   RUNG wire#w2
      Contact( "Flag".MV06_Auto )
   END_RUNG wire#w4
   RUNG wire#w1
      I_Contact( "Allarm".MV_06_FAULT )
      wire#w5
      Contact( "Flag".MV06_Auto )
      wire#w6
      Contact( "MV06 PID UP" )
      wire#w7
      I_Contact( "Close MV06" )
      I_Contact( "Inputs".MV06_Open )
      Coil( "Open MV06" )
   END_RUNG
   RUNG wire#w6
      Contact( "Shot to open" )
   END_RUNG wire#w7
   RUNG wire#w5
      Contact( "Flag".MV06_Open )
      wire#w8
      Contact( "MV WORK PULSE" )
   END_RUNG wire#w7
   RUNG wire#w8
      Contact( "ON" )
   END_RUNG wire#w7
   RUNG wire#w5
      Contact( "Flag".MV06_Auto )
      wire#w9
      Contact( "MV06 PID DOWN" )
      wire#w10
      I_Contact( "Open MV06" )
      I_Contact( "Inputs"."MV06 Close" )
      Coil( "Close MV06" )
   END_RUNG
   RUNG wire#w9
      Contact( "Shot to close" )
   END_RUNG wire#w10
   RUNG wire#w5
      Contact( "Flag".MV06_Close )
      wire#w11
      Contact( "MV WORK PULSE" )
   END_RUNG wire#w10
   RUNG wire#w11
      Contact( "ON" )
   END_RUNG wire#w10
   // the same network as SCL:
   #_w1 := NOT "ON" AND NOT "ON";
   IF #_w1 AND ("Inputs".MV06_Open OR "Flag".MV06_Close OR "Flag".MV06_Auto) THEN
       "Flag".MV06_Open := FALSE;
   END_IF;
   IF #_w1 AND ("Inputs"."MV06 Close" OR "Flag".MV06_Open OR "Flag".MV06_Auto) THEN
       "Flag".MV06_Close := FALSE;
   END_IF;
   #_w2 := NOT "ON" AND NOT "Allarm".MV_06_FAULT;
   "Open MV06" := #_w2 AND (("Flag".MV06_Auto AND ("MV06 PID UP" OR "Shot to open")) OR ("Flag".MV06_Open AND ("MV WORK PULSE" OR "ON"))) AND NOT "Close MV06" AND NOT "Inputs".MV06_Open;
   "Close MV06" := #_w2 AND (("Flag".MV06_Auto AND ("MV06 PID DOWN" OR "Shot to close")) OR ("Flag".MV06_Close AND ("MV WORK PULSE" OR "ON"))) AND NOT "Open MV06" AND NOT "Inputs"."MV06 Close";
END_REGION

REGION Network 11: Motorized valve work time pulse generator
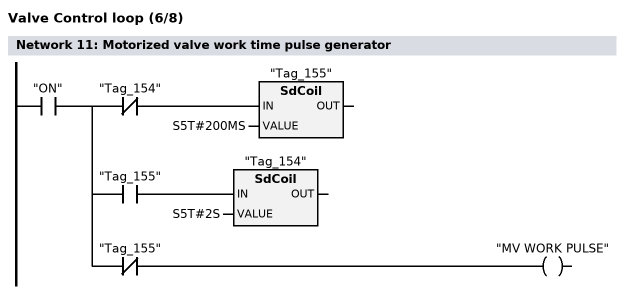
   // no SCL statement known for SdCoil: written as a call
   #_w1 := "ON";
   SdCoil(in := "ON" AND NOT "Tag_154", value := S5T#200MS, operand := "Tag_155");
   SdCoil(in := #_w1 AND "Tag_155", value := S5T#2S, operand := "Tag_154");
   "MV WORK PULSE" := #_w1 AND NOT "Tag_155";
END_REGION

REGION Network 12: Motorized valve pulse generator for rotation control
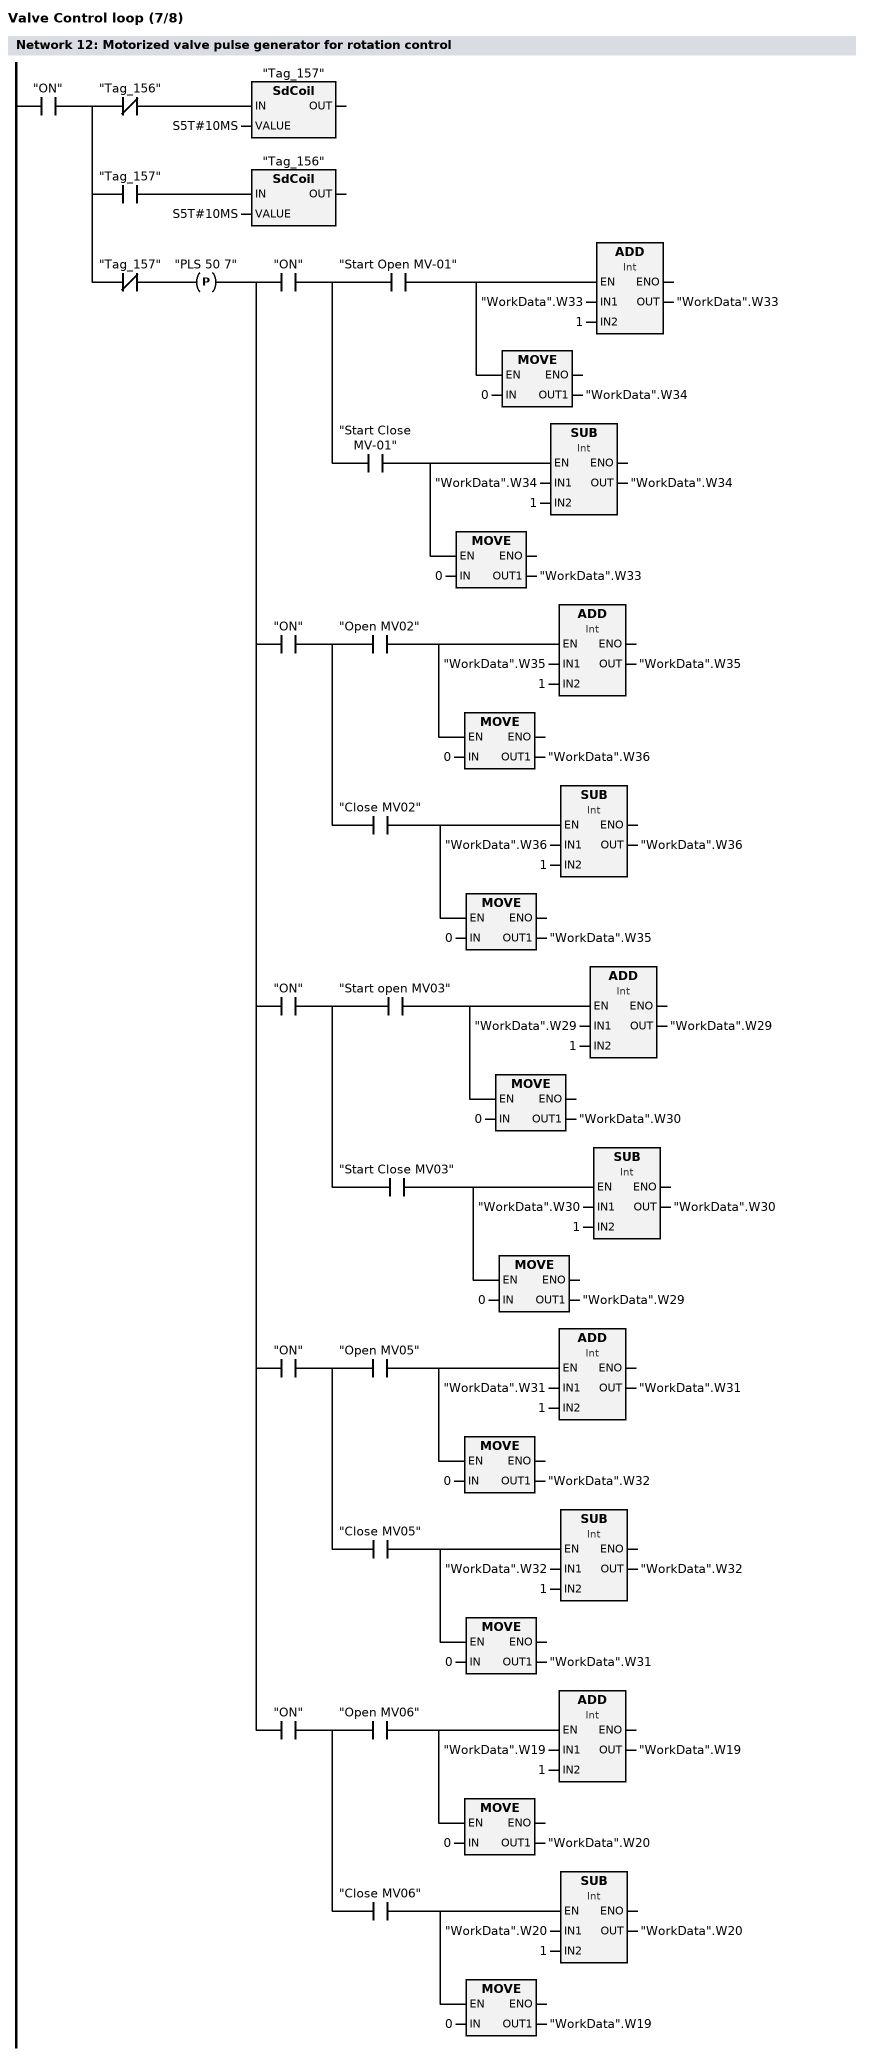
   // no SCL statement known for SdCoil: written as a call
   #_w1 := "ON";
   SdCoil(in := "ON" AND NOT "Tag_156", value := S5T#10MS, operand := "Tag_157");
   SdCoil(in := #_w1 AND "Tag_157", value := S5T#10MS, operand := "Tag_156");
   #_w2 := #_w1 AND NOT "Tag_157";
   #_w3 := #_w2 AND NOT "PLS 50 7";   // rising edge
   "PLS 50 7" := #_w2;
   #_w4 := #_w3 AND "ON";
   IF #_w4 AND "Start Open MV-01" THEN
       "WorkData".W33 := "WorkData".W33 + 1;
       "WorkData".W34 := 0;
   END_IF;
   IF #_w4 AND "Start Close MV-01" THEN
       "WorkData".W34 := "WorkData".W34 - 1;
       "WorkData".W33 := 0;
   END_IF;
   #_w5 := #_w3 AND "ON";
   IF #_w5 AND "Open MV02" THEN
       "WorkData".W35 := "WorkData".W35 + 1;
       "WorkData".W36 := 0;
   END_IF;
   IF #_w5 AND "Close MV02" THEN
       "WorkData".W36 := "WorkData".W36 - 1;
       "WorkData".W35 := 0;
   END_IF;
   #_w6 := #_w3 AND "ON";
   IF #_w6 AND "Start open MV03" THEN
       "WorkData".W29 := "WorkData".W29 + 1;
       "WorkData".W30 := 0;
   END_IF;
   IF #_w6 AND "Start Close MV03" THEN
       "WorkData".W30 := "WorkData".W30 - 1;
       "WorkData".W29 := 0;
   END_IF;
   #_w7 := #_w3 AND "ON";
   IF #_w7 AND "Open MV05" THEN
       "WorkData".W31 := "WorkData".W31 + 1;
       "WorkData".W32 := 0;
   END_IF;
   IF #_w7 AND "Close MV05" THEN
       "WorkData".W32 := "WorkData".W32 - 1;
       "WorkData".W31 := 0;
   END_IF;
   #_w8 := #_w3 AND "ON";
   IF #_w8 AND "Open MV06" THEN
       "WorkData".W19 := "WorkData".W19 + 1;
       "WorkData".W20 := 0;
   END_IF;
   IF #_w8 AND "Close MV06" THEN
       "WorkData".W20 := "WorkData".W20 - 1;
       "WorkData".W19 := 0;
   END_IF;
END_REGION

REGION Network 13: Verify theorical valve position for out of range / Motorized valve fault
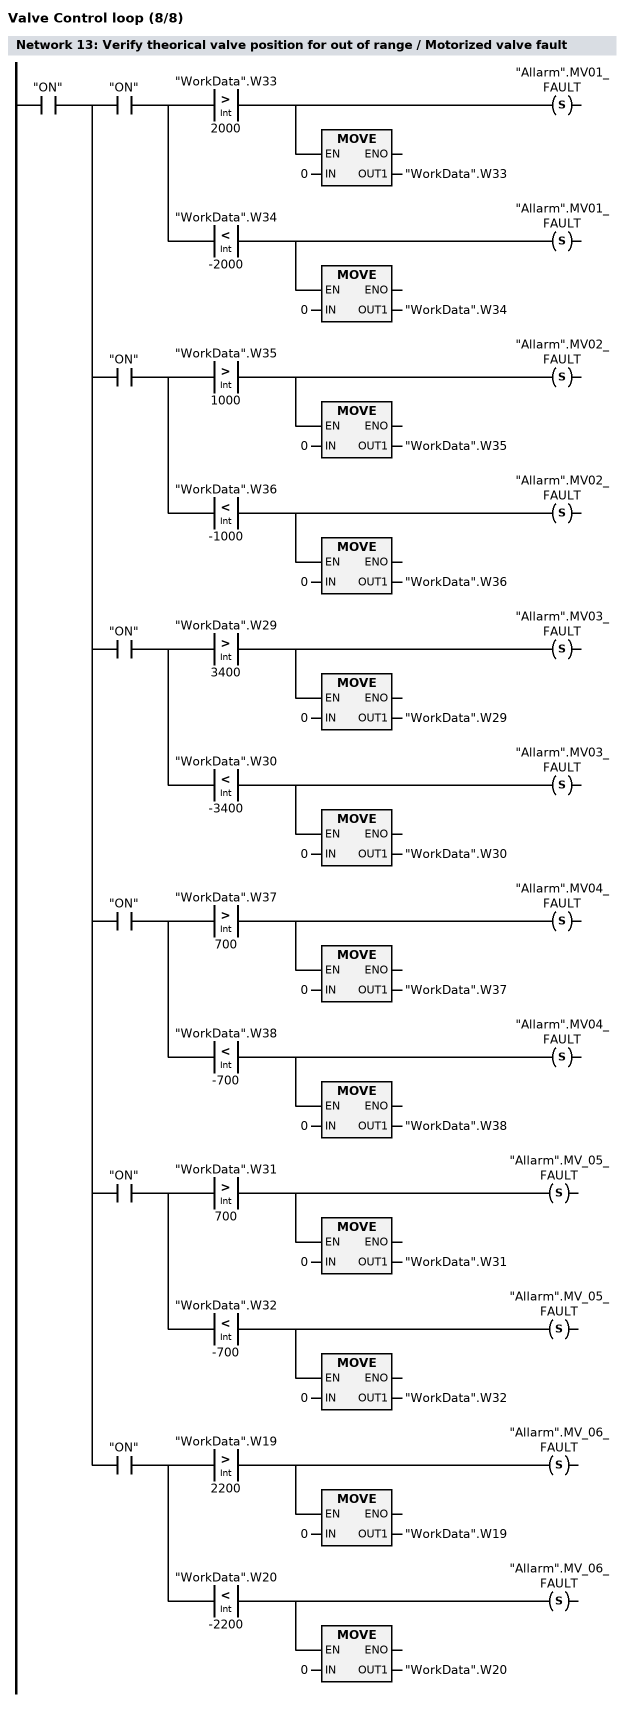
   RUNG wire#powerrail
      Contact( "ON" )
      wire#w1
      Contact( "ON" )
      wire#w2
      { S7_Templates := "SrcType := Int" } GT_Contact(in1 := "WorkData".W33, in2 := 2000)
      wire#w3
      S_Coil( "Allarm".MV01_FAULT )
   END_RUNG
   RUNG wire#w3
      { S7_GenerateENO := "TRUE" } Move(in := 0, out1 => "WorkData".W33)
   END_RUNG
   RUNG wire#w2
      { S7_Templates := "SrcType := Int" } LT_Contact(in1 := "WorkData".W34, in2 := -2000)
      wire#w4
      S_Coil( "Allarm".MV01_FAULT )
   END_RUNG
   RUNG wire#w4
      { S7_GenerateENO := "TRUE" } Move(in := 0, out1 => "WorkData".W34)
   END_RUNG
   RUNG wire#w1
      Contact( "ON" )
      wire#w5
      { S7_Templates := "SrcType := Int" } GT_Contact(in1 := "WorkData".W35, in2 := 1000)
      wire#w6
      S_Coil( "Allarm".MV02_FAULT )
   END_RUNG
   RUNG wire#w6
      { S7_GenerateENO := "TRUE" } Move(in := 0, out1 => "WorkData".W35)
   END_RUNG
   RUNG wire#w5
      { S7_Templates := "SrcType := Int" } LT_Contact(in1 := "WorkData".W36, in2 := -1000)
      wire#w7
      S_Coil( "Allarm".MV02_FAULT )
   END_RUNG
   RUNG wire#w7
      { S7_GenerateENO := "TRUE" } Move(in := 0, out1 => "WorkData".W36)
   END_RUNG
   RUNG wire#w1
      Contact( "ON" )
      wire#w8
      { S7_Templates := "SrcType := Int" } GT_Contact(in1 := "WorkData".W29, in2 := 3400)
      wire#w9
      S_Coil( "Allarm".MV03_FAULT )
   END_RUNG
   RUNG wire#w9
      { S7_GenerateENO := "TRUE" } Move(in := 0, out1 => "WorkData".W29)
   END_RUNG
   RUNG wire#w8
      { S7_Templates := "SrcType := Int" } LT_Contact(in1 := "WorkData".W30, in2 := -3400)
      wire#w10
      S_Coil( "Allarm".MV03_FAULT )
   END_RUNG
   RUNG wire#w10
      { S7_GenerateENO := "TRUE" } Move(in := 0, out1 => "WorkData".W30)
   END_RUNG
   RUNG wire#w1
      Contact( "ON" )
      wire#w11
      { S7_Templates := "SrcType := Int" } GT_Contact(in1 := "WorkData".W37, in2 := 700)
      wire#w12
      S_Coil( "Allarm".MV04_FAULT )
   END_RUNG
   RUNG wire#w12
      { S7_GenerateENO := "TRUE" } Move(in := 0, out1 => "WorkData".W37)
   END_RUNG
   RUNG wire#w11
      { S7_Templates := "SrcType := Int" } LT_Contact(in1 := "WorkData".W38, in2 := -700)
      wire#w13
      S_Coil( "Allarm".MV04_FAULT )
   END_RUNG
   RUNG wire#w13
      { S7_GenerateENO := "TRUE" } Move(in := 0, out1 => "WorkData".W38)
   END_RUNG
   RUNG wire#w1
      Contact( "ON" )
      wire#w14
      { S7_Templates := "SrcType := Int" } GT_Contact(in1 := "WorkData".W31, in2 := 700)
      wire#w15
      S_Coil( "Allarm".MV_05_FAULT )
   END_RUNG
   RUNG wire#w15
      { S7_GenerateENO := "TRUE" } Move(in := 0, out1 => "WorkData".W31)
   END_RUNG
   RUNG wire#w14
      { S7_Templates := "SrcType := Int" } LT_Contact(in1 := "WorkData".W32, in2 := -700)
      wire#w16
      S_Coil( "Allarm".MV_05_FAULT )
   END_RUNG
   RUNG wire#w16
      { S7_GenerateENO := "TRUE" } Move(in := 0, out1 => "WorkData".W32)
   END_RUNG
   RUNG wire#w1
      Contact( "ON" )
      wire#w17
      { S7_Templates := "SrcType := Int" } GT_Contact(in1 := "WorkData".W19, in2 := 2200)
      wire#w18
      S_Coil( "Allarm".MV_06_FAULT )
   END_RUNG
   RUNG wire#w18
      { S7_GenerateENO := "TRUE" } Move(in := 0, out1 => "WorkData".W19)
   END_RUNG
   RUNG wire#w17
      { S7_Templates := "SrcType := Int" } LT_Contact(in1 := "WorkData".W20, in2 := -2200)
      wire#w19
      S_Coil( "Allarm".MV_06_FAULT )
   END_RUNG
   RUNG wire#w19
      { S7_GenerateENO := "TRUE" } Move(in := 0, out1 => "WorkData".W20)
   END_RUNG
   // the same network as SCL:
   #_w1 := "ON" AND "ON";
   IF #_w1 AND ("WorkData".W33 > 2000) THEN
       "Allarm".MV01_FAULT := TRUE;
       "WorkData".W33 := 0;
   END_IF;
   IF #_w1 AND ("WorkData".W34 < (-2000)) THEN
       "Allarm".MV01_FAULT := TRUE;
       "WorkData".W34 := 0;
   END_IF;
   #_w2 := "ON" AND "ON";
   IF #_w2 AND ("WorkData".W35 > 1000) THEN
       "Allarm".MV02_FAULT := TRUE;
       "WorkData".W35 := 0;
   END_IF;
   IF #_w2 AND ("WorkData".W36 < (-1000)) THEN
       "Allarm".MV02_FAULT := TRUE;
       "WorkData".W36 := 0;
   END_IF;
   #_w3 := "ON" AND "ON";
   IF #_w3 AND ("WorkData".W29 > 3400) THEN
       "Allarm".MV03_FAULT := TRUE;
       "WorkData".W29 := 0;
   END_IF;
   IF #_w3 AND ("WorkData".W30 < (-3400)) THEN
       "Allarm".MV03_FAULT := TRUE;
       "WorkData".W30 := 0;
   END_IF;
   #_w4 := "ON" AND "ON";
   IF #_w4 AND ("WorkData".W37 > 700) THEN
       "Allarm".MV04_FAULT := TRUE;
       "WorkData".W37 := 0;
   END_IF;
   IF #_w4 AND ("WorkData".W38 < (-700)) THEN
       "Allarm".MV04_FAULT := TRUE;
       "WorkData".W38 := 0;
   END_IF;
   #_w5 := "ON" AND "ON";
   IF #_w5 AND ("WorkData".W31 > 700) THEN
       "Allarm".MV_05_FAULT := TRUE;
       "WorkData".W31 := 0;
   END_IF;
   IF #_w5 AND ("WorkData".W32 < (-700)) THEN
       "Allarm".MV_05_FAULT := TRUE;
       "WorkData".W32 := 0;
   END_IF;
   #_w6 := "ON" AND "ON";
   IF #_w6 AND ("WorkData".W19 > 2200) THEN
       "Allarm".MV_06_FAULT := TRUE;
       "WorkData".W19 := 0;
   END_IF;
   IF #_w6 AND ("WorkData".W20 < (-2200)) THEN
       "Allarm".MV_06_FAULT := TRUE;
       "WorkData".W20 := 0;
   END_IF;
END_REGION
END_FUNCTION

FUNCTION "Analog output conversion" : Void   // FC18, LAD
TITLE = Analog output
{ S7_Optimized_Access := 'FALSE' }
VERSION : 0.1
   VAR_TEMP
      App00 : DInt;
      App01 : DInt;
      App03 : DInt;
      App04 : DInt;
      app05 : DInt;
      Calcolo_Aria : Int;
      Correzione_Aria : Int;
      Consegna_Motorino_Aria : Int;
      test_out : DInt;
      Prod_h : Real;
      tmp : Real;
   END_VAR
   VAR_TEMP   // added for the SCL form of the ladder/FBD networks
      _w1 : Bool;
   END_VAR
BEGIN

REGION Network 1: Plant limits
